Staubli VAL3: HOME.pjx

--- HOME.pjx ---
Parameters version=s7.7 stackSize=5000 millimeterUnit=true
Program file=checkPoint.pgx
Program file=checkZone.pgx
Program file=computeFrame.pgx
Program file=delete.pgx
Program file=deleteItem.pgx
Program file=duplicate.pgx
Program file=find.pgx
Program file=findMove.pgx
Program file=get.pgx
Program file=getDistance.pgx
Program file=getFrame.pgx
Program file=getFrameId.pgx
Program file=getFunctionEdit.pgx
Program file=getFunctionSel.pgx
Program file=getFunctionView.pgx
Program file=getJointData.pgx
Program file=getListItem.pgx
Program file=getMoveType.pgx
Program file=getPoint.pgx
Program file=getPointData.pgx
Program file=getSize.pgx
Program file=getSizeItem.pgx
Program file=getTool.pgx
Program file=getTrajItem.pgx
Program file=getTrajType.pgx
Program file=goTo.pgx
Program file=HerePoint.pgx
Program file=insertItem.pgx
Program file=insertValue.pgx
Program file=interpolateJ.pgx
Program file=link_me.pgx
Program file=listAdd.pgx
Program file=load.pgx
Program file=loadCycle.pgx
Program file=loadJoint.pgx
Program file=loadPage.pgx
Program file=loadPoint.pgx
Program file=makeTraj.pgx
Program file=moveTo.pgx
Program file=new.pgx
Program file=onEdit.pgx
Program file=onEditItem.pgx
Program file=onFunctionEdit.pgx
Program file=onFunctionSel.pgx
Program file=onFunctionView.pgx
Program file=onInsert.pgx
Program file=onProgEnd.pgx
Program file=onRun.pgx
Program file=onSave.pgx
Program file=onStart.pgx
Program file=onStop.pgx
Program file=orderDistance.pgx
Program file=orderZone.pgx
Program file=page_changeTrsf.pgx
Program file=scan_bestFit.pgx
Program file=select.pgx
Program file=selectProg.pgx
Program file=selectZone.pgx
Program file=setFrameId.pgx
Program file=setPointFrame.pgx
Program file=setTool.pgx
Program file=setTrajItem.pgx
Data file=HOME.dtx
Library alias=saveData path=Disk://saveData/saveData.pjx
Library alias=page path=Disk://kernel/template/page/page.pjx
Library alias=use path=Disk://kernel/userPage/userPage.pjx
Library alias=cycleStatus path=Disk://cycleStatus/cycleStatus.pjx
Library alias=language path=Disk://kernel/language/language.pjx
Library alias=tcp path=Disk://kernel/tool/tool.pjx
Library alias=prog path=Disk://instruction/PROG/PROG.pjx
Library alias=processList path=Disk://kernel/processList/processList.pjx
Library alias=solid path=Disk://trajectory/check_solid/check_solid.pjx
Library alias=pt path=Disk://kernel/template/session/saveTraj/HOME/HOME.pjx
Type name=TrajectoryItem path=Disk://kernel/template/TrajectoryItem/TrajectoryItem.pjx
Type name=ActionItem path=Disk://kernel/template/ActionItem/ActionItem.pjx
Type name=InstrItem path=Disk://kernel/template/InstrItem/InstrItem.pjx
Type name=Trajectory path=Disk://kernel/template/Trajectory/Trajectory.pjx
Type name=trajectoryType path=Disk://kernel/template/trajectory/trajectory.pjx
Type name=TrajHome path=Disk://kernel/template/TrajHome/TrajHome.pjx
Type name=TrajJoint path=Disk://kernel/template/TrajJoint/TrajJoint.pjx
Type name=TrajPoint path=Disk://kernel/template/TrajPoint/TrajPoint.pjx
Type name=FrameItem path=Disk://kernel/template/FrameItem/FrameItem.pjx

--- HOME.dtx ---
InstrItem tcpInstr
  [0]
    string sType
    string sData
Trajectory tTraj
  [0]
    TrajectoryItem tSuper[3]
      [0]
        num distance
        num moveType
        num nTime
        num nStop
        num nTcpAction
        string comment
        bool toStop
        mdesc nom_speed = {tmax=300, rmax=9999, leave=30, reach=30}
        InstrItem iInstr[3]
          [0]
            string sType
            string sData
          [1]
            string sType
            string sData
          [2]
            string sType
            string sData
        num nMoveId
      [1]
        num distance
        num moveType
        num nTime
        num nStop
        num nTcpAction
        string comment = "@JPOINT jZone1"
        bool toStop
        mdesc nom_speed = {tmax=9999, rmax=9999, leave=30, reach=30}
        InstrItem iInstr[3]
          [0]
            string sType
            string sData
          [1]
            string sType
            string sData
          [2]
            string sType
            string sData
        num nMoveId
      [2]
        num distance
        num moveType = 1
        num nTime
        num nStop
        num nTcpAction
        string comment = "@JPOINT jZone1Out"
        bool toStop
        mdesc nom_speed = {vel=450, tmax=1500, rmax=9999, leave=30, reach=30}
        InstrItem iInstr[3]
          [0]
            string sType
            string sData
          [1]
            string sType
            string sData
          [2]
            string sType
            string sData
        num nMoveId
    string sID = "HOME Zone1"
    num nId
public bool bMoveType[3]
  [0] = true
  [1] = true
public bool bStepping
bool bToSave
frame fFrame = {fatherId=world[0]}
frame fSetFrame = {x=-364.286321, y=-1043.316491, z=11.196424, rx=-6.99985, ry=11.31473, rz=18.24134, fatherId=world[0]}
mdesc nom_speed = {accel=25, vel=25, decel=25, blend=off}
num nCoeff = 1
num nDistance = 357.24033
num nHome
num nIndex
num nJoint
num nKey
num nSelected
num nView
num nZeta
pointRx pBestFit[3]
  [0] = {fatherId=world[0]}
  [1] = {fatherId=world[0]}
  [2] = {fatherId=world[0]}
pointRx pCheck = {fatherId=world[0]}
pointRx pNull = {fatherId=world[0]}
pointRx pPointTo = {fatherId=world[0]}
pointRx pPoints[3]
  [0] = {x=-364.286321, y=-1043.316491, z=11.196424, rx=84.453459, ry=18.310573, rz=168.800057, shoulder=lefty, elbow=epositive, wrist=wnegative, fatherId=world[0]}
  [1] = {x=-169.661081, y=-983.133224, z=-35.427424, rx=84.45454, ry=18.311675, rz=168.800636, shoulder=lefty, elbow=epositive, wrist=wnegative, fatherId=world[0]}
  [2] = {x=-263.249747, y=-701.832631, z=-51.099539, rx=84.453256, ry=18.310748, rz=168.801333, shoulder=lefty, elbow=epositive, wrist=wnegative, fatherId=world[0]}
string sInstruction
string sInstruction2
public string sItems[7]
  [0] = "cube_Salle_Bl"
  [1] = "cube_evac_rebut"
  [2] = "cube_moule"
  [3] = "cube_prelev"
  [4] = "home"
string sJoint = "Pt_Pass_Centre"
string sJointCycle = "Pt_Pass_Centre"
string sList
string sMessage
string sPoint = "Centre_Moule"
string sPointCycle = "Centre_Moule"
string sTrajType = "HOME"
trsf tAppro
trsf tPointTo
mdesc mMdesc = {accel=10, vel=10, decel=10, blend=off}
TrajHome jEditPoint
  [0]
    num nIndexTool
    TrajJointItem tData
      [0]
        jointRx jJoint
        TrajectoryItem tSuper
          [0]
            num distance
            num moveType
            num nTime
            num nStop
            num nTcpAction
            string comment
            bool toStop
            mdesc nom_speed = {accel=50, vel=50, decel=50, tmax=300, rmax=9999, leave=30, reach=30}
            InstrItem iInstr[3]
              [0]
                string sType
                string sData
              [1]
                string sType
                string sData
              [2]
                string sType
                string sData
            num nMoveId
    string sID
    num nZoneType
    num nZoneMove
    pointRx pO
    pointRx pX
    pointRx pY
    num nDimension
    pointRx pPointMove
    frame fFrame
    string sProgram
    num nIndexFrame
string sTrajCycle

--- checkPoint.pgx ---
public program checkPoint(point x_PointToGo (dimensions=1), point x_PointStart (dimensions=1), bool& x_bUnreached[] (dimensions=1), tool x_tTool (dimensions=1), bool x_bLinear (dimensions=1))
  local joint jPoint
  local string message
  local num i
  local trsf t
begin
  // check if the point is null
  if (cycleStatus:bCycle==false and cycleStatus:bSimulation==false) or !x_bLinear
    x_bUnreached=false
    t=position(x_PointToGo,world)
    if t!={0,0,0,0,0,0}
      //
      // look if the point that you want to reach is valid
      if x_bLinear
        //
        // use the percentage....
        //
        for i=0.1 to 1 step 0.1
          pCheck.trsf=interpolateL(position(x_PointStart,world),position(x_PointToGo,world),i)
          x_bUnreached=!pointToJoint(x_tTool,herej(),pCheck,jPoint)
          if x_bUnreached
            return
          endIf
        endFor
      else
        // joint move or check only the working area
        x_PointToGo.config={sfree,efree,wfree}
        x_bUnreached=!pointToJoint(x_tTool,herej(),x_PointToGo,jPoint)
      endIf
    endIf
  endIf
end

--- checkZone.pgx ---
program checkZone(point& x_pPoints[] (dimensions=1), tool x_tTool (dimensions=1), num x_nDimension (dimensions=1), num x_nType (dimensions=1), bool& x_bInside (dimensions=1))
begin
  // init the variable
  x_bInside=false
  // show the frame
  switch x_nType
    case 1
      //
      // BOX
      //
      //create the cube
      call solid:create_cube(x_pPoints[0],x_pPoints[1],x_pPoints[2],x_nDimension)
      // check the cube
      call solid:check_cube(x_tTool,x_bInside)
    break
    case 2
      //
      // SPHERE
      //
      // create the sphere
      call solid:create_sphere(x_pPoints,x_nDimension)
      // check the cube
      call solid:check_sphere(x_tTool,x_bInside)
    break
    case 3
      //
      // PLANE
      //
      //create the plane
      call solid:create_plane(x_pPoints[0],x_pPoints[1],x_pPoints[2])
      // check the cube
      call solid:check_plane(x_tTool,x_bInside)
    break
  endSwitch
end

--- delete.pgx ---
public program delete(string x_sName, num& x_nResult[])
  local string l_sItem
  local num l_nSize
  local string l_sMessage
begin
  //
  // delete the select trajectory
  //
  if isDefined(pt:tTraj[x_sName]) and x_sName!="home"
    // delete
    delete(pt:tTraj[x_sName])
    // save it
    bToSave=true
    x_nResult=0
  elseIf x_sName=="home"
    call language:message(l_sMessage,133)
    popUpMsg(l_sMessage)
  else
    x_nResult=-1
  endIf
end

--- findMove.pgx ---
program findMove(num x_nIndex, tool x_tTool, num& x_nMoveType[])
  local point l_pHere
  local num l_nResult
  local num l_nIndexTool
  local num l_nSize
  local num l_nMoveType
  local point l_pPoint[2]
  local joint l_jHere
  local bool l_bUnreach
begin
  //
  // MOVE TO THE POINT
  //
  // use the flange
  x_tTool=flange
  // get all the value that you need
  l_nSize=size(jEditPoint.tData)
  l_pHere=here(x_tTool,world)
  // get the point and the circle point
  call getPoint(l_pPoint,false,x_nIndex)
  pPoints[1].trsf=position(l_pPoint,world)
  pPoints[2].trsf={0,0,0,0,0,0}
  // Set to JOINT for default
  x_nMoveType=0
  // get the move TYPE
  call getMoveType(l_nMoveType,x_nIndex,false)
  //
  // move forward
  //
  if x_nIndex>0 and l_nMoveType==1
    // get the point and the circle point
    call getPoint(l_pPoint,false,x_nIndex-1)
    pPoints.trsf=position(l_pPoint,world)
    if distance(l_pHere,pPoints)<25
      // set to linear
      x_nMoveType=1
    elseIf setFrame(pPoints,pPoints[1],pPoints[2],fSetFrame)==0
      // check frame
      l_pHere=here(x_tTool,fSetFrame)
      pPoints[1].trsf=position(pPoints[1],fSetFrame)
      if l_pHere.trsf.x>=0 and l_pHere.trsf.x<=pPoints[1].trsf.x and abs(l_pHere.trsf.y)<10 and abs(l_pHere.trsf.z)<10
        // set to linear
        x_nMoveType=1
      endIf
    endIf
  endIf
  //
  // move back
  //
  if x_nIndex<(l_nSize-1) and x_nMoveType!=1
    call getMoveType(l_nMoveType,x_nIndex+1,false)
    if l_nMoveType==1
      // get the point and the circle point
      call getPoint(l_pPoint,false,x_nIndex)
      pPoints[1].trsf=position(l_pPoint,world)
      // get the point and the circle point
      call getPoint(l_pPoint,false,x_nIndex+1)
      pPoints.trsf=position(l_pPoint,world)
      if distance(l_pHere,pPoints)<25
        // switch to linear
        x_nMoveType=1
      elseIf setFrame(pPoints,pPoints[1],pPoints[2],fSetFrame)==0
        // check frame
        l_pHere=here(x_tTool,fSetFrame)
        pPoints[1].trsf=position(pPoints[1],fSetFrame)
        if l_pHere.trsf.x>=0 and l_pHere.trsf.x<=pPoints[1].trsf.x and abs(l_pHere.trsf.y)<10 and abs(l_pHere.trsf.z)<10
          // set to linear
          x_nMoveType=1
        endIf
      endIf
    endIf
  endIf
end

--- getFrame.pgx ---
public program getFrame(frame& x_fFrame[], bool x_bCycle)
  local num l_nIndex
begin
  // CYCLE
  if x_bCycle
    l_nIndex=pt:tTraj[sTrajCycle].nIndexFrame
  else
    // NOT CYCLE
    l_nIndex=jEditPoint.nIndexFrame
  endIf
  x_fFrame.trsf=saveData:fFrameItem[l_nIndex].fFrame.trsf
end

--- getFrameId.pgx ---
public program getFrameId(num& x_nFrame)
begin
  // give back the frame
  x_nFrame=jEditPoint.nIndexFrame
end

--- getFunctionEdit.pgx ---
public program getFunctionEdit(string& x_sName[])
  local string l_sMessage
begin
  //
  // define your message for the
  // function KEY
  //
  // NOTE is an ARRAY[0..7]
  //
  // example:
  // x_sName[1]="DEMO"
  // active the F2 button
  //
  if (nIndex>0 or jEditPoint.nZoneType==0) and find(jEditPoint.tData[nIndex].tSuper.comment,"@")==-1
    // here
    call language:message(l_sMessage,150)
    x_sName[0]=l_sMessage
  else
  // ALIGN
  call language:message(l_sMessage,134)
  x_sName[1]=l_sMessage
  // Tool
  call language:message(l_sMessage,123)
  x_sName[2]=l_sMessage
  endIf
//  // define the @Link
//  x_sName[1]="@Link"
end

--- getFunctionSel.pgx ---
public program getFunctionSel(string& x_sName[])
  local string l_sMessage
begin
  //
  // define your message for the
  // function KEY
  //
  // NOTE is an ARRAY[0..7]
  //
  // example:
  // x_sName[1]="DEMO"
  // active the F2 button
  //
  // Set Home Program
  call language:message(l_sMessage,135)
  x_sName[2]=l_sMessage
  call language:message(l_sMessage,136)
  x_sName[3]=l_sMessage
end

--- getFunctionView.pgx ---
public program getFunctionView(string& x_sName[])
  local string l_sMessage
begin
  //
  // define your message for the
  // function KEY
  //
  // NOTE is an ARRAY[0..7]
  //
  // example:
  // x_sName[1]="DEMO"
  // active the F2 button
  //
  // define the @Link
  // here
  call language:message(l_sMessage,150)
  x_sName[0]=l_sMessage
  // x_sName[1]="@Link"
    // ALIGN
  call language:message(l_sMessage,134)
  x_sName[1]=l_sMessage
end

--- getJointData.pgx ---
public program getJointData(joint& x_jJoint, tool& x_tTool, bool x_bCycle, num x_nIndex)
  local point l_pPoint
  local num l_nSize
  local string l_sName
  local num l_nResult
  local string l_sComment
  local num l_nType
  local point l_pPointTo
  local num i
begin
  //
  //   !!! REMOVE DUE PROBLEMS of CROSS LINK
  //
  //   get the comment type
  //    if x_bCycle
  //      l_sComment=pt:tTraj[sTrajCycle].tData[x_nIndex].tSuper.comment
  //    else
  //      l_sComment=jEditPoint.tData[x_nIndex].tSuper.comment
  //    endIf
  //    if find(l_sComment,"@POINT")!=-1
  //      //
  //      // POINT
  //      //
  //      l_sName=right(l_sComment,len(l_sComment)-len("@POINT "))
  //      call loadPoint(l_sName,l_nResult)
  //      if l_nResult==0
  //        // use the flange
  //        x_tTool=flange
  //        // get the tool
  //        //call tcp:getTool(x_tTool,pPoint:tTraj[l_sName].nIndexTool)
  //        // get the last point using the depart point
  //        l_nSize=size(pPoint:tTraj[l_sName].tData)
  //        // find the point use the real one
  //        for i=0 to l_nSize-1
  //          l_nType=pPoint:tTraj[l_sName].tData[i].nType
  //          if l_nType==1
  //            // get the real point
  //            l_pPointTo=pPoint:tTraj[l_sName].tData[i].pPoint
  //          endIf
  //        endFor
  //        // take the DEPART
  //        l_pPoint=pPoint:tTraj[l_sName].tData[l_nSize-1].pPoint
  //        l_pPoint=appro(l_pPointTo,l_pPoint.trsf)
  //        // give back
  //        pointToJoint(x_tTool,herej(),l_pPoint,x_jJoint)
  //      endIf
  //    elseIf find(l_sComment,"@JPOINT")!=-1
  //      //
  //      // JPOINT
  //      //
  //      l_sName=right(l_sComment,len(l_sComment)-len("@JPOINT "))
  //      call loadJoint(l_sName,l_nResult)
  //      if l_nResult==0
  //        // use the flange
  //        x_tTool=flange
  //        // give back
  //        //call tcp:getTool(x_tTool,jPoint:tTraj[l_sName].nIndexTool)
  //        x_jJoint=jPoint:tTraj[l_sName].tData[0].jJoint
  //      endIf
  //    else
  // give back
  // use the flange
  x_tTool=flange
  if x_bCycle
    x_jJoint=pt:tTraj[sTrajCycle].tData[x_nIndex].jJoint
    //      call tcp:getTool(x_tTool,pt:tTraj[sTrajCycle].nIndexTool)
  else
    x_jJoint=jEditPoint.tData[x_nIndex].jJoint
    //      call tcp:getTool(x_tTool,jEditPoint.nIndexTool)
  endIf
  //endIf
  if l_nResult!=0
    // remove the link
    jEditPoint.tData[x_nIndex].tSuper.comment=""
  endIf
end

--- getListItem.pgx ---
public program getListItem(string& x_sItem[], num x_nIndex)
  local string l_sItem4[4]
  local string l_sZoneType
  local string l_sZoneMove
  local string l_sItem7[7]
  local joint l_jJoint
  local tool l_tTool
  local string l_sItem[6]
begin
  //
  // define the item to show in the edit page Traj
  // customize an array and copy to x_sItem...
  //
  // see other traj as example
  l_sItem[0]=l_sItem7[0]=("Joint 1 > "+toString(".2",jEditPoint.tData[x_nIndex].jJoint.j1))
  l_sItem[1]=l_sItem7[1]=("Joint 2 > "+toString(".2",jEditPoint.tData[x_nIndex].jJoint.j2))
  l_sItem[2]=l_sItem7[2]=("Joint 3 > "+toString(".2",jEditPoint.tData[x_nIndex].jJoint.j3))
  l_sItem[3]=l_sItem7[3]=("Joint 4 > "+toString(".2",jEditPoint.tData[x_nIndex].jJoint.j4))
  l_sItem[4]=l_sItem7[4]=("Joint 5 > "+toString(".2",jEditPoint.tData[x_nIndex].jJoint.j5))
  l_sItem[5]=l_sItem7[5]=("Joint 6 > "+toString(".2",jEditPoint.tData[x_nIndex].jJoint.j6))
  call use:stringCopy(l_sItem,x_sItem)
  switch x_nIndex
    case 0
      // add_on for the zone definition
      switch jEditPoint.nZoneType
        case 1
          l_sZoneType=" > Box"
        break
        case 2
          l_sZoneType=" > Sphere"
        break
        case 3
          l_sZoneType=" > Plane"
        break
        default
          l_sZoneType=" > "
        break
      endSwitch
      // show only the necessary
      if jEditPoint.nZoneType[x_nIndex]==0
        l_sItem7[6]=("Zone "+l_sZoneType)
        call use:stringCopy(l_sItem7,x_sItem)
      else
        // only the move type
        l_sItem4[0]=("Zone "+l_sZoneType)
        switch jEditPoint.nZoneMove
          case 0
            l_sZoneMove="Point"
          break
          case 1
            l_sZoneMove="Appro"
          break
          case 2
            l_sZoneMove="Z Value"
          break
          case 3
            l_sZoneMove="@Point"
          break
          case 4
            l_sZoneMove="@JPoint"
          break
        endSwitch
        l_sItem4[1]="  └───>[EDIT] "
        l_sItem4[2]=("MoveTO > "+l_sZoneMove)
        if (jEditPoint.nZoneMove==3 or jEditPoint.nZoneMove==4) and find(jEditPoint.tData.tSuper.comment,"@")!=-1
          l_sItem4[3]="  └> "+jEditPoint.tData.tSuper.comment
        else
          l_sItem4[3]="  └───>[EDIT] "
        endIf
        // insert all
        call use:stringCopy(l_sItem4,x_sItem)
      endIf
    break
    default
      // insert only the coordinate
      call use:stringCopy(l_sItem,x_sItem)
    break
  endSwitch
  // save the actual index
  nIndex=x_nIndex
end

--- getMoveType.pgx ---
public program getMoveType(num& x_nMoveType[], num x_nIndex, bool x_bCycle)
begin
  // get the moveType
  if x_bCycle
    x_nMoveType=pt:tTraj[sTrajCycle].tData[x_nIndex].tSuper.moveType
  else
    x_nMoveType=jEditPoint.tData[x_nIndex].tSuper.moveType
  endIf
end

--- getPoint.pgx ---
public program getPoint(point& x_pPoint[] (dimensions=1), bool x_bCycle (dimensions=1), num x_nIndex (dimensions=1))
  local string l_sItem
  local tool l_tTool
  local joint l_jJoint
begin
  // check the point
  link(x_pPoint,world)
  // use the flange
  l_tTool=flange
  // give back the point
  call getJointData(l_jJoint,l_tTool,x_bCycle,x_nIndex)
  x_pPoint=jointToPoint(l_tTool,world,l_jJoint)
end

--- getPointData.pgx ---
program getPointData(num& x_nSpeed[], mdesc& x_mDesc[], num& x_nDistance[], bool& x_bToStop[], num& x_nMoveType[], num& x_nStop[], num x_nIndex, bool x_bCycle)
begin
  if x_bCycle
    // get tha parameter
    // SPEED
    // get the speed in mm/sec
    if pt:tTraj[sTrajCycle].tData[x_nIndex].tSuper.moveType==0
      x_nSpeed=pt:tTraj[sTrajCycle].tData[x_nIndex].tSuper.nom_speed.vel*15
    else
      if pt:tTraj[sTrajCycle].tData[x_nIndex].tSuper.moveType==1
        x_nSpeed=pt:tTraj[sTrajCycle].tData[x_nIndex].tSuper.nom_speed.tvel
      endIf
    endIf
    // MDESC
    x_mDesc=pt:tTraj[sTrajCycle].tData[x_nIndex].tSuper.nom_speed
    // DISTANCE
    x_nDistance=pt:tTraj[sTrajCycle].tData[x_nIndex].tSuper.distance
    //  check  for a stop using
    x_bToStop=pt:tTraj[sTrajCycle].tData[x_nIndex].tSuper.toStop
    // get MoveType
    x_nMoveType=pt:tTraj[sTrajCycle].tData[x_nIndex].tSuper.moveType
  else
    // get tha parameter
    // SPEED
    // get the speed in mm/sec
    if jEditPoint.tData[x_nIndex].tSuper.moveType==0
      x_nSpeed=jEditPoint.tData[x_nIndex].tSuper.nom_speed.vel*15
    else
      if jEditPoint.tData[x_nIndex].tSuper.moveType==1
        x_nSpeed=jEditPoint.tData[x_nIndex].tSuper.nom_speed.tvel
      endIf
    endIf
    // MDESC
    x_mDesc=jEditPoint.tData[x_nIndex].tSuper.nom_speed
    // DISTANCE
    x_nDistance=jEditPoint.tData[x_nIndex].tSuper.distance
    //  check  for a stop using
    x_bToStop=jEditPoint.tData[x_nIndex].tSuper.toStop
    // get MoveType
    x_nMoveType=jEditPoint.tData[x_nIndex].tSuper.moveType
  endIf
end

--- getSize.pgx ---
public program getSize(num& x_nSize[])
  local string l_sType
begin
  // give back the size to trajectory field
  x_nSize=size(pt:tTraj)
end

--- getTool.pgx ---
public program getTool(num& x_nTool)
begin
  //
  // get the tool
  //
  x_nTool=jEditPoint.nIndexTool
end

--- getTrajItem.pgx ---
public program getTrajItem(TrajectoryItem& x_tTrajItem[], num x_nIndex)
begin
  //
  // get all the FIELD
  //
  x_tTrajItem=jEditPoint.tData[x_nIndex].tSuper
end

--- getTrajType.pgx ---
program getTrajType(string& x_sTrajType[])
  local num l_nPos
  local string l_sPath
begin
  // get the trajType
  l_sPath=libPath()
  if find(l_sPath,sTrajType)==-1
    do
      l_nPos=find(l_sPath,"/")
      if l_nPos==-1
        l_nPos=find(l_sPath,"\")
      endIf
      if l_nPos!=-1
        l_sPath=right(l_sPath,len(l_sPath)-l_nPos-1)
      endIf
    until l_nPos==-1
    //
    sTrajType=l_sPath
  endIf
  // return back
  x_sTrajType=sTrajType
end

--- goTo.pgx ---
public program goTo(tool x_tTool, mdesc x_mDesc, num x_nMoveType, bool& x_bUnreached[], num x_nIndex)
  local mdesc temp_mdesc
  local num l_nSize
  local point l_pPoint
  local joint l_jJoint
  local frame l_ZoneFrame
  local bool l_bCheck
  local num l_nType
  local num l_nDimension
  local tool l_tTool
  local string l_sMessage
  local num l_nMoveId
begin
  // check for the zone
  if (jEditPoint.nZoneType!=0 and x_nIndex==0) or find(jEditPoint.tData[x_nIndex].tSuper.comment,"@")!=-1
    // take the tool
    // use flange
    l_tTool=flange
    //call tcp:getTool(l_tTool,jEditPoint.nIndexTool)
    // take the three points
    pPoints[0]=jEditPoint.pO
    pPoints[1]=jEditPoint.pX
    pPoints[2]=jEditPoint.pY
    // take the distance
    l_nDimension=jEditPoint.nDimension
    //take the type
    l_nType=jEditPoint.nZoneType
    // check the frame type-2 CIRCLE
    if setFrame(pPoints[0],pPoints[1],pPoints[2],fSetFrame)==0 or l_nType==2
      call checkZone(pPoints,l_tTool,l_nDimension,l_nType,l_bCheck)
      // show the result
      if l_bCheck
        // inside the zone
        call language:message(l_sMessage,225)
        // move TO
        call moveTo(l_tTool,x_mDesc,x_nMoveType,x_bUnreached,x_nIndex,l_nMoveId,false)
      elseIf find(jEditPoint.tData[x_nIndex].tSuper.comment,"@")!=-1
        // link POINT
        // look for the moveType
        call findMove(x_nIndex,l_tTool,x_nMoveType)
        call moveTo(l_tTool,x_mDesc,x_nMoveType,x_bUnreached,x_nIndex,l_nMoveId,false)
      else
        //outside the zone
        call language:message(l_sMessage,226)
      endIf
    elseIf find(jEditPoint.tData[x_nIndex].tSuper.comment,"@")!=-1
      // found a @POINT-JPOINT
      call moveTo(l_tTool,x_mDesc,x_nMoveType,x_bUnreached,x_nIndex,l_nMoveId,false)
    else
      // frame not define
      call language:message(l_sMessage,183)
      call use:timerDialog(l_sMessage,3)
    endIf
  elseIf isInRange(jEditPoint.tData[x_nIndex].jJoint)
    // look for the moveType
    call findMove(x_nIndex,x_tTool,x_nMoveType)
    // execute the movement
    switch x_nMoveType
      case 0
        // JOINT MOVE
        // go to the select Joint
        movej(jEditPoint.tData[x_nIndex].jJoint,x_tTool,x_mDesc)
      break
      case 1
        // LINEAR MOVE
        movel(jointToPoint(x_tTool,world,jEditPoint.tData[x_nIndex].jJoint),x_tTool,x_mDesc)
      break
      default
      break
    endSwitch
  else
    x_bUnreached=true
  endIf
  // save the actual index
  nIndex=x_nIndex
end

--- insertValue.pgx ---
program insertValue(num& x_nValue[] (dimensions=1), num x_nIndex (dimensions=1))
begin
  if nDistance[0]!=-1
    // insert
    insert(nDistance[x_nIndex])
    insert(nCoeff[x_nIndex])
    insert(nJoint[x_nIndex])
    insert(nHome[x_nIndex])
  endIf
  // copy
  nCoeff[x_nIndex]=x_nValue[3]
  nDistance[x_nIndex]=x_nValue[2]
  nJoint[x_nIndex]=x_nValue[1]
  nHome[x_nIndex]=x_nValue
end

--- interpolateJ.pgx ---
public program interpolateJ(joint p_j1, joint p_j2, num p_nInterpolate, joint& x_jRetVal[], bool& x_bRetVal[])
begin
  // Interpolierten Jointwert berechnen
  x_jRetVal.j1=(p_j2.j1-p_j1.j1)*p_nInterpolate+p_j1.j1
  x_jRetVal.j2=(p_j2.j2-p_j1.j2)*p_nInterpolate+p_j1.j2
  x_jRetVal.j3=(p_j2.j3-p_j1.j3)*p_nInterpolate+p_j1.j3
  x_jRetVal.j4=(p_j2.j4-p_j1.j4)*p_nInterpolate+p_j1.j4
  x_jRetVal.j5=(p_j2.j5-p_j1.j5)*p_nInterpolate+p_j1.j5
  x_jRetVal.j6=(p_j2.j6-p_j1.j6)*p_nInterpolate+p_j1.j6
  x_bRetVal=isInRange(x_jRetVal)
end

--- link_me.pgx ---
program link_me(num x_nIndex)
  local num i
  local num l_nSize
  local string l_sItem
  local num l_nKey
  local num l_nIndex
  local string l_sEvent
begin
  //
  // !!! REMOVE DUE PROBLEMS of CROSS LINK
  //
  //  // @POINT -> use depart
  //  // @JOINT -> use the first JOINT
  //  call use:clear(0,13)
  //  call use:type(5,13,"@Link")
  //  call use:setSizeList(4,8,8,3)
  //  call use:listcreate("")
  //  l_sItem=" NONE "
  //  call use:listadd(l_sItem)
  //  l_sItem="@JPOINT"
  //  call use:listadd(l_sItem)
  //  //  l_sItem="@POINT"
  //  //  call use:listadd(l_sItem)
  //  // refresh it
  //  call use:listupdate(0)
  //  // get the item
  //  do
  //    l_nKey=get()
  //    call use:listevent(l_nKey,l_nIndex,l_sEvent)
  //  until l_nKey==270 or l_nKey==255
  //  if l_nKey==270
  //    // select the @Point - @jPoint
  //    // build the list
  //    call use:setSizeList(0,0,16,12)
  //    switch l_nIndex
  //      case 2
  //        call use:listcreate("@Point")
  //        // insert all the item
  //        l_sItem=first(pPoint:tTraj)
  //        call use:listadd(l_sItem)
  //        // search it
  //        while l_sItem!=""
  //          l_sItem=next(pPoint:tTraj[l_sItem])
  //          call use:listadd(l_sItem)
  //        endWhile
  //        l_sItem="@POINT "
  //      break
  //      case 1
  //        call use:listcreate("@JPoint")
  //        // insert all the item
  //        l_sItem=first(jPoint:tTraj)
  //        call use:listadd(l_sItem)
  //        // search it
  //        while l_sItem!=""
  //          l_sItem=next(jPoint:tTraj[l_sItem])
  //          call use:listadd(l_sItem)
  //        endWhile
  //        l_sItem="@JPOINT "
  //      break
  //      case 0
  //        // empty one
  //        l_sItem=l_sEvent=""
  //      break
  //    endSwitch
  //    if l_nIndex!=0
  //      // refresh it
  //      call use:listupdate(0)
  //      // get the item
  //      do
  //        l_nKey=get()
  //        call use:listevent(l_nKey,l_nIndex,l_sEvent)
  //      until l_nKey==270 or l_nKey==255
  //    endIf
  //    // give back
  //    if l_nKey==270
  //      // save it
  //      jEditPoint.tData[x_nIndex].tSuper.comment=l_sItem+l_sEvent
  //      if x_nIndex==0
  //        jEditPoint.nZoneType=0
  //      endIf
  //    endIf
  //  endIf
end

--- load.pgx ---
public program load(string x_sItem, num& x_nResult)
  local string l_sType
  local string l_sPath
  local string l_sMessage
begin
  // load the select trajectory..already loaded
  call getTrajType(l_sType)
  if find(pt:libPath(),saveData:sPathTraj)==-1
    pt:libLoad(saveData:sPathTraj+l_sType)
    delay(0)
    if saveData:bDebug
      ? "loading HOME..."+saveData:sPathTraj+l_sType
    endIf
  endIf
  if isDefined(pt:tTraj[x_sItem])
    // use the type...
    call pt:link_it(x_sItem)
    jEditPoint=pt:tTraj[x_sItem]
    jEditPoint.sID=x_sItem
    x_nResult=0
  elseIf x_sItem!=""
    // not FOUND
    call language:message(l_sMessage,-7)
    x_nResult=-1
    popUpMsg(l_sMessage+x_sItem)
    jEditPoint.sID=""
  elseIf x_sItem==""
    // reload all the template
    call loadJoint("",x_nResult)
    call loadPoint("",x_nResult)
  endIf
end

--- loadCycle.pgx ---
public program loadCycle(string x_sItem, num& x_nResult[])
  local string l_sType
  local string l_sPath
begin
  // load the select trajectory..already loaded
  call getTrajType(l_sType)
  if find(pt:libPath(),saveData:sPathTraj)==-1
    pt:libLoad(saveData:sPathTraj+l_sType)
    delay(0)
  endIf
  if isDefined(pt:tTraj[x_sItem])
    // use the type...
    call pt:link_it(x_sItem)
    sTrajCycle=x_sItem
  else
    x_nResult=-1
  endIf
end

--- loadJoint.pgx ---
public program loadJoint(string x_sItem, num& x_nResult)
  local string l_sType
  local string l_sMessage
  local num l_nResult
begin
  //
  // !!! REMOVE DUE PROBLEMS of CROSS LINK
  //
  //
  //  // load the select trajectory..already loaded
  //  call getTrajType(l_sType)
  //  if find(jPoint:libPath(),saveData:sPathTraj)==-1
  //    l_nResult=jPoint:libLoad(saveData:sPathTraj+"JPOINT")
  //    delay(0)
  //    if saveData:bDebug
  //      ? "HOME loading JPOINT..."+saveData:sPathTraj+"JPOINT"+toString("",l_nResult)
  //    endIf
  //  endIf
  //  if isDefined(jPoint:tTraj[x_sItem])
  //    // validate
  //    x_nResult=0
  //  elseIf x_sItem!=""
  //    // not FOUND
  //    call language:message(l_sMessage,-7)
  //    x_nResult=-1
  //    popUpMsg(l_sMessage+x_sItem)
  //  endIf
end

--- loadPage.pgx ---
program loadPage(string x_sPage, string& x_sItems[])
// load the next page
  local num i
begin
  // look if the page libload is correct
  i=page:libLoad(x_sPage)
  delay(0)
  logMsg("KERNEL:PAGE LIBLOAD "+x_sPage+" result "+toString("",i))
  if i!=0
    popUpMsg("Loading page "+x_sPage+" error CODE "+toString("",i))
  else
    page:sItems=x_sItems
    call page:main()
  endIf
end

--- loadPoint.pgx ---
public program loadPoint(string x_sItem, num& x_nResult)
  local string l_sType
  local string l_sMessage
  local num l_nResult
begin
  //
  // !!! REMOVE DUE PROBLEMS of CROSS LINK
  //
  //  // load the select trajectory..already loaded
  //  call getTrajType(l_sType)
  //  if find(pPoint:libPath(),saveData:sPathTraj)==-1
  //    l_nResult=pPoint:libLoad(saveData:sPathTraj+"POINT")
  //    delay(0)
  //    if saveData:bDebug
  //      ? "HOME loading POINT..."+saveData:sPathTraj+"POINT"+toString("",l_nResult)
  //    endIf
  //  endIf
  //  if isDefined(pPoint:tTraj[x_sItem])
  //    // validate
  //    x_nResult=0
  //  elseIf x_sItem!=""
  //    // not FOUND
  //    call language:message(l_sMessage,-7)
  //    x_nResult=-1
  //    popUpMsg(l_sMessage+x_sItem)
  //  endIf
end

--- makeTraj.pgx ---
program makeTraj(num x_nJointStart, string x_sTrajLoad)
  local num i
  local bool l_bToStop[2]
  local num l_nSize
  local tool l_tTool
  local num l_nSpeed[2]
  local mdesc l_mDesc[2]
  local num l_nDistance[2]
  local num l_nMoveType[2]
  local point l_pAction
  local bool l_bUnreached
  local num l_nStop
  local point l_pCheck[3]
  local point l_pHere
  local frame l_fPlane
  local num l_nTime
  local string l_sType
  local string l_sMessage
  local bool l_bConnection
  local num l_nMoveId
  local TrajectoryItem l_tTraj
  local joint l_jJoint
  local ActionItem l_aAction
  local num j
  local bool l_bGoToCloseP
  local point l_pHereJ
  local joint l_jResult
  local bool l_bOk
  local num i_from
  local num i_to
  local joint l_jHere
  local joint l_jRunJoint[2]
begin
  //
  // inizialize the system
  //
  // use the flange
  l_tTool=flange
  // the maximum size
  call getSizeItem(true,l_nSize)
  //
  // first go near by straight line of the two previous points
  //
  if pt:tTraj[sTrajCycle].nZoneType!=0 and x_nJointStart==0
    // use of the ZONE TYPE
    switch pt:tTraj[sTrajCycle].nZoneMove
      case 0
        l_sType="POINT"
      break
      case 1
        l_sType="APPRO"
      break
      case 2
        l_sType="Z VALUE"
      break
      case 3
        l_sType="@Point"
      break
      case 4
        l_sType="@JPoint"
      break
    endSwitch
    cycleStatus:sToShow="Move using: "+l_sType+toString("",x_nJointStart)+"# of the home: "+x_sTrajLoad
    logMsg("HOMING: "+l_sMessage)
    call getPointData(l_nSpeed,l_mDesc,l_nDistance,l_bToStop,l_nMoveType,l_nStop,0,true)
    call moveTo(l_tTool,l_mDesc,l_nMoveType,l_bUnreached,0,l_nMoveId,true)
    waitEndMove()
    // set the start point
    x_nJointStart=1
  elseIf saveData:bUseHomeScanner
    // look FORWARD
    if x_nJointStart<l_nSize-1
      // get all the JOINT
      call getJointData(l_jRunJoint[0],l_tTool,true,x_nJointStart+1)
      call getJointData(l_jRunJoint[1],l_tTool,true,x_nJointStart)
      // look if there is
      if setFrame(jointToPoint(l_tTool,world,l_jRunJoint[0]),jointToPoint(l_tTool,world,l_jRunJoint[1]),pNull,fFrame)==0
        pCheck=here(l_tTool,fFrame)
        if pCheck.trsf.x>=0
          //
          // go to nearest point
          //
          call getPoint(l_pCheck[0],true,x_nJointStart+1)
          call getPoint(l_pCheck[1],true,x_nJointStart)
          x_nJointStart=x_nJointStart+1
          l_bGoToCloseP=true
        endIf
      endIf
    endIf
    // LOOK BACKWARD
    if !l_bGoToCloseP and x_nJointStart>0
      // get all the JOINT
      call getJointData(l_jRunJoint[0],l_tTool,true,x_nJointStart)
      call getJointData(l_jRunJoint[1],l_tTool,true,x_nJointStart-1)
      // look if there is
      if setFrame(jointToPoint(l_tTool,world,l_jRunJoint[0]),jointToPoint(l_tTool,world,l_jRunJoint[1]),pNull,fFrame)==0
        pCheck=here(l_tTool,fFrame)
        if pCheck.trsf.x>=0
          //
          // go to nearest point
          //
          call getPoint(l_pCheck[0],true,x_nJointStart)
          call getPoint(l_pCheck[1],true,x_nJointStart-1)
          l_bGoToCloseP=true
        endIf
      endIf
    endIf
    // go to an approach POINT
    if l_bGoToCloseP
      // init
      l_pCheck[2]=here(l_tTool,world)
      l_pHere=here(l_tTool,world)
      l_pHereJ=here(flange,world)
      l_nDistance=10000
      // check the nearest point
      l_nMoveType=pt:tTraj[sTrajCycle].tData[x_nJointStart].tSuper.moveType
      for i=0 to 1 step 0.1
        if l_nMoveType==0
          call interpolateJ(l_jRunJoint[1],l_jRunJoint[0],i,l_jResult,l_bOk)
          l_pCheck[2]=jointToPoint(flange,world,l_jResult)
          if l_nDistance>=distance(l_pCheck[2],l_pHereJ)
            l_nDistance=distance(l_pCheck[2],l_pHereJ)
            //save the value
            l_nStop=i
          endIf
        else
          l_pCheck[2].trsf=interpolateL(l_pCheck[1].trsf,l_pCheck[0].trsf,i)
          l_bOk=true
          if l_nDistance>=distance(l_pCheck[2],l_pHere)
            l_nDistance=distance(l_pCheck[2],l_pHere)
            //save the value
            l_nStop=i
          endIf
        endIf
      endFor
      // closer search
      i_from=(max(l_nStop-0.05,0))
      i_to=(min(l_nStop+0.05,1))
      for i=i_from to i_to step 0.01
        if l_nMoveType==0
          call interpolateJ(l_jRunJoint[1],l_jRunJoint[0],i,l_jResult,l_bOk)
          l_pCheck[2]=jointToPoint(flange,world,l_jResult)
          if l_nDistance>=distance(l_pCheck[2],l_pHereJ)
            l_nDistance=distance(l_pCheck[2],l_pHereJ)
            //save the value
            l_nStop=i
          endIf
        else
          l_pCheck[2].trsf=interpolateL(l_pCheck[1].trsf,l_pCheck[0].trsf,i)
          l_bOk=true
          if l_nDistance>=distance(l_pCheck[2],l_pHere)
            l_nDistance=distance(l_pCheck[2],l_pHere)
            //save the value
            l_nStop=i
          endIf
        endIf
      endFor
      // set the best one
      call getPointData(l_nSpeed,l_mDesc,l_nDistance,l_bToStop,l_nMoveType,l_nStop,x_nJointStart,true)
      l_jHere=herej()
      if l_nMoveType==0
        call interpolateJ(l_jRunJoint[1],l_jRunJoint[0],l_nStop,l_jResult,l_bOk)
        l_pCheck[2]=jointToPoint(flange,world,l_jResult)
        // put the wrist on free
        l_pCheck[2].config.wrist=wfree
        if pointToJoint(l_tTool,herej(),l_pCheck[2],l_jHere)
          movej(l_pCheck[2],flange,l_mDesc)
        endIf
      else
        l_pCheck[2].trsf=interpolateL(l_pCheck[1].trsf,l_pCheck[0].trsf,l_nStop)
        // put the wrist on free
        l_pCheck[2].config.wrist=wfree
        if pointToJoint(l_tTool,herej(),l_pCheck[2],l_jHere)
          movej(l_pCheck[2],l_tTool,l_mDesc)
        endIf
      endIf
      // show the message
      cycleStatus:sToShow="Move to point: "+toString("",x_nJointStart+1)+" of: "+x_sTrajLoad +" % "+toString(".3",l_nStop)
      logMsg("HOMING: "+cycleStatus:sToShow)
      waitEndMove()
    endIf
  endIf
  //
  // for all of my traj cyclePoints move the robot
  //
  resize(tTraj.tSuper,1,size(pt:tTraj[sTrajCycle].tData))
  for i=x_nJointStart to (l_nSize-1)
    tTraj.tSuper[i]=pt:tTraj[sTrajCycle].tData[i].tSuper
  endFor
  tTraj.sID="HOME "+pt:tTraj[sTrajCycle].sID
  call cycleStatus:addTraj(tTraj)
  // show the message
  cycleStatus:sToShow="Moving from point: "+toString("",x_nJointStart+1)+" of : "+x_sTrajLoad
  logMsg("HOMING: "+cycleStatus:sToShow)
  for i=x_nJointStart to (l_nSize-1)
    //
    // get the point info
    //
    l_tTraj=pt:tTraj[sTrajCycle].tData[i].tSuper
    //
    // get the distance in percentage
    //
    call getDistance(l_tTool,l_nDistance,true,i)
    //
    // give to the traj library the percentage distance
    //
    if l_tTraj.toStop
      l_tTraj.nom_speed.blend=off
    endIf
    //
    // put the move in the stack
    //
    l_jJoint=pt:tTraj[sTrajCycle].tData[i].jJoint
    call moveTo(l_tTool,l_tTraj.nom_speed,l_tTraj.moveType,l_bUnreached,i,l_nMoveId,true)
    // set the data
    l_aAction.nDistance=l_nDistance
    l_aAction.nPointId=i
    l_aAction.nMoveId=l_nMoveId
    l_aAction.sIdTraj="HOME "+pt:tTraj[sTrajCycle].sID
    call cycleStatus:putInstr_Traj(l_aAction,l_tTraj,pt:tTraj[sTrajCycle].nIndexTool,l_nSize)
    // there is a waitEndMove
    if l_tTraj.toStop
      waitEndMove()
      delay(l_tTraj.nStop)
      // wait all the action has been done
      wait(cycleStatus:bActionRunning==false)
    endIf
  endFor
end

--- moveTo.pgx ---
public program moveTo(tool x_tTool, mdesc x_mDesc, num x_nMoveType, bool& x_bUnreached[], num x_nIndex, num& x_nMoveId, bool x_bCycle)
  local frame l_fFrame
  local point l_pHere
  local point l_pMove
  local string l_sName
  local num i
  local num l_nType
  local num l_nIndex
  local num l_nResult
  local joint l_jMove
  local num l_nSize
  local tool l_tTool
  local point l_pPoint
begin
  if x_bCycle
    //
    // go to the select Joint
    //
    // use the go to the defined type...
    if x_nIndex==0 and pt:tTraj[sTrajCycle].nZoneType!=0
      switch pt:tTraj[sTrajCycle].nZoneMove
        // POINT TO
        case 0
          if x_nMoveType==0
            x_nMoveId=movej(pt:tTraj[sTrajCycle].pPointMove,x_tTool,x_mDesc)
          elseIf x_nMoveType==1
            x_nMoveId=movel(pt:tTraj[sTrajCycle].pPointMove,x_tTool,x_mDesc)
          endIf
        break
        case 1
          // APPRO use the real APPRO
          call tcp:getTool(l_tTool,pt:tTraj[sTrajCycle].nIndexTool)
          if x_nMoveType==0
            x_nMoveId=movej(appro(here(l_tTool,world),pt:tTraj[sTrajCycle].pPointMove.trsf),x_tTool,x_mDesc)
          elseIf x_nMoveType==1
            x_nMoveId=movel(appro(here(l_tTool,world),pt:tTraj[sTrajCycle].pPointMove.trsf),x_tTool,x_mDesc)
          endIf
        break
        case 2
          // Z VALUE
          if pt:tTraj[sTrajCycle].fFrame.trsf!={0,0,0,0,0,0}
            l_pHere=here(x_tTool,pt:tTraj[sTrajCycle].fFrame)
            l_pHere.trsf.z=pt:tTraj[sTrajCycle].pPointMove.trsf.z
            if x_nMoveType==0
              x_nMoveId=movej(l_pHere,x_tTool,x_mDesc)
            elseIf x_nMoveType==1
              x_nMoveId=movel(l_pHere,x_tTool,x_mDesc)
            endIf
          endIf
        break
        case 3,4
          // @POINT @JPOINT
          call getJointData(l_jMove,l_tTool,x_bCycle,x_nIndex)
          // MOVE
          if x_nMoveType==0
            x_nMoveId=movej(l_jMove,x_tTool,x_mDesc)
          elseIf x_nMoveType==1
            l_pPoint=jointToPoint(x_tTool,world,l_jMove)
            l_pPoint.config={ssame,esame,wsame}
            x_nMoveId=movel(l_pPoint,x_tTool,x_mDesc)
          endIf
        break
      endSwitch
    else
      // get the JOINT DATA
      call getJointData(l_jMove,l_tTool,x_bCycle,x_nIndex)
      // MOVE
      if x_nMoveType==0
        x_nMoveId=movej(l_jMove,l_tTool,x_mDesc)
      elseIf x_nMoveType==1
        l_pPoint=jointToPoint(l_tTool,world,l_jMove)
        l_pPoint.config={ssame,esame,wsame}
        x_nMoveId=movel(l_pPoint,l_tTool,x_mDesc)
      endIf
    endIf
  else
    //
    // go to the select Joint
    //
    // use the go to the defined type...
    if x_nIndex==0 and jEditPoint.nZoneType!=0
      switch jEditPoint.nZoneMove
        // POINT TO
        case 0
          if x_nMoveType==0
            x_nMoveId=movej(jEditPoint.pPointMove,x_tTool,x_mDesc)
          elseIf x_nMoveType==1
            x_nMoveId=movel(jEditPoint.pPointMove,x_tTool,x_mDesc)
          endIf
        break
        case 1
          // APPRO gat the tool taught
          call tcp:getTool(l_tTool,jEditPoint.nIndexTool)
          if x_nMoveType==0
            x_nMoveId=movej(appro(here(l_tTool,world),jEditPoint.pPointMove.trsf),x_tTool,x_mDesc)
          elseIf x_nMoveType==1
            x_nMoveId=movel(appro(here(l_tTool,world),jEditPoint.pPointMove.trsf),x_tTool,x_mDesc)
          endIf
        break
        case 2
          // Z VALUE
          if jEditPoint.fFrame.trsf!={0,0,0,0,0,0}
            l_pHere=here(x_tTool,jEditPoint.fFrame)
            l_pHere.trsf.z=jEditPoint.pPointMove.trsf.z
            if x_nMoveType==0
              x_nMoveId=movej(l_pHere,x_tTool,x_mDesc)
            elseIf x_nMoveType==1
              x_nMoveId=movel(l_pHere,x_tTool,x_mDesc)
            endIf
          endIf
        break
        case 3,4
          // get the JOINT DATA
          call getJointData(l_jMove,l_tTool,x_bCycle,x_nIndex)
          // MOVE
          if x_nMoveType==0
            x_nMoveId=movej(l_jMove,x_tTool,x_mDesc)
          elseIf x_nMoveType==1
            l_pPoint=jointToPoint(x_tTool,world,l_jMove)
            l_pPoint.config={ssame,esame,wsame}
            x_nMoveId=movel(l_pPoint,x_tTool,x_mDesc)
          endIf
        break
      endSwitch
    else
      // get the JOINT DATA
      call getJointData(l_jMove,l_tTool,x_bCycle,x_nIndex)
      // MOVE
      if x_nMoveType==0
        x_nMoveId=movej(l_jMove,l_tTool,x_mDesc)
      elseIf x_nMoveType==1
        l_pPoint=jointToPoint(l_tTool,world,l_jMove)
        l_pPoint.config={ssame,esame,wsame}
        x_nMoveId=movel(l_pPoint,l_tTool,x_mDesc)
      endIf
    endIf
  endIf
end

--- new.pgx ---
public program new(string x_sName, num& x_nResult[])
  local string l_sPrefix
  local num l_nResult
begin
  // new one
  if insert(pt:tTraj[x_sName])
    call pt:link_it(x_sName)
    pt:tTraj[x_sName].nIndexTool=saveData:nIndexTool
    x_nResult=0
    // set it
    bToSave=true
  else
    x_nResult=-1
  endIf
end

--- onEdit.pgx ---
public program onEdit(string& x_sItem[])
  local string l_sPath
  local string l_sName
  local num l_nResult
begin
  // DEFINE YOUR ITEM
  call getTrajType(saveData:sTrajTypeUsing)
  // load the trajectory
  call load(x_sItem,l_nResult)
  if size(x_sItem)>1
    // give back the path
    l_sPath="Disk://trajectory/page_viewTraj"
    x_sItem[1]=x_sItem
    x_sItem=l_sPath
    // init
    tAppro={0,0,0,0,0,0}
    tPointTo={0,0,0,0,0,0}
    nZeta=0
  endIf
end

--- onEditItem.pgx ---
public program onEditItem(string& x_sEvent[], num x_nIndex, num x_nIndexItem)
  local joint l_jJoint
  local num i
  local string l_sMessage
  local string l_sEmpty
  local string l_sItem5[5]
  local num l_nMin
  local num l_nMax
  local num l_nValue
  local trsf l_tNull
  local tool l_tTool
  local point l_pPoint
  local num l_nSize
  local num l_nKey
  local num l_nIndex
  local string l_sEvent
  local string l_sItem[4]
begin
  // edit the custom element that was add in the list
  l_jJoint=jEditPoint.tData[x_nIndexItem].jJoint
  call use:findPos(x_sEvent,">",i)
  i=i+1
  // clean the line
  call use:listcursor(use:nView,false)
  l_sEmpty=""
  if x_nIndexItem>0 or (jEditPoint.nZoneType[x_nIndexItem]==0)
    if find(jEditPoint.tData[x_nIndexItem].tSuper.comment,"@")==-1 and (jEditPoint.nZoneType==0 or x_nIndexItem>0)
      switch x_nIndex
        case 0
          //  j1-value
          if cycleStatus:bCycle
            // set a limit +- 5
            call use:changeValue(l_jJoint.j1,l_jJoint.j1-5,l_jJoint.j1+5,i+40-use:nBottomX,use:nView+1,l_sEmpty)
          else
            call use:changeValue(l_jJoint.j1,0,0,i+40-use:nBottomX,use:nView+1,l_sEmpty)
          endIf
        break
        case 1
          //  j2-value
          if cycleStatus:bCycle
            // set a limit +- 5
            call use:changeValue(l_jJoint.j2,l_jJoint.j2-5,l_jJoint.j2+5,i+40-use:nBottomX,use:nView+1,l_sEmpty)
          else
            call use:changeValue(l_jJoint.j2,0,0,i+40-use:nBottomX,use:nView+1,l_sEmpty)
          endIf
        break
        case 2
          //  j3-value
          if cycleStatus:bCycle
            // set a limit +- 5
            call use:changeValue(l_jJoint.j3,l_jJoint.j3-5,l_jJoint.j3+5,i+40-use:nBottomX,use:nView+1,l_sEmpty)
          else
            call use:changeValue(l_jJoint.j3,0,0,i+40-use:nBottomX,use:nView+1,l_sEmpty)
          endIf
        break
        case 3
          //  j4-value
          if cycleStatus:bCycle
            // set a limit +- 5
            call use:changeValue(l_jJoint.j4,l_jJoint.j4-5,l_jJoint.j4+5,i+40-use:nBottomX,use:nView+1,l_sEmpty)
          else
            call use:changeValue(l_jJoint.j4,0,0,i+40-use:nBottomX,use:nView+1,l_sEmpty)
          endIf
        break
        case 4
          //  j5-value
          if cycleStatus:bCycle
            // set a limit +- 5
            call use:changeValue(l_jJoint.j5,l_jJoint.j5-5,l_jJoint.j5+5,i+40-use:nBottomX,use:nView+1,l_sEmpty)
          else
            call use:changeValue(l_jJoint.j5,0,0,i+40-use:nBottomX,use:nView+1,l_sEmpty)
          endIf
        break
        case 5
          //  j6-value
          if cycleStatus:bCycle
            // set a limit +- 5
            call use:changeValue(l_jJoint.j6,l_jJoint.j6-5,l_jJoint.j6+5,i+40-use:nBottomX,use:nView+1,l_sEmpty)
          else
            call use:changeValue(l_jJoint.j6,0,0,i+40-use:nBottomX,use:nView+1,l_sEmpty)
          endIf
        break
      endSwitch
    endIf
    switch x_nIndex
      case 6
        // change the move type
        l_sItem="---"
        l_sItem[1]="Box"
        l_sItem[2]="Sphere"
        l_sItem[3]="Plane"
        call use:clear(0,13)
        call use:changeValue(jEditPoint.nZoneType[x_nIndexItem],0,0,i+40-use:nBottomX,use:nView+1,l_sItem)
      break
    endSwitch
  elseIf x_nIndexItem==0
    switch x_nIndex
      // change the MOVE-TYPE
      case 0
        l_sItem[0]=" - - - "
        l_sItem[1]="Box"
        l_sItem[2]="Sphere"
        l_sItem[3]="Plane"
        call use:clear(0,13)
        call use:changeValue(jEditPoint.nZoneType,0,0,i+40-use:nBottomX,use:nView+1,l_sItem)
      break
      // edit the MOVE-TYPE
      case 1
        switch jEditPoint.nZoneType
          case 1
            // BOX
            call setPointFrame(jEditPoint.fFrame.trsf,jEditPoint.pO,jEditPoint.pX,jEditPoint.pY,jEditPoint.nDimension,1)
            if jEditPoint.fFrame.trsf=={0,0,0,0,0,0}
              call use:timerDialog("the frame has NOT been teached",2)
            endIf
          break
          case 2
            // sphere
            call page_changeTrsf(jEditPoint.pO.trsf,"Sphere"," teach the origin...",true,jEditPoint.nDimension,"radius",world)
            jEditPoint.pX=compose(jEditPoint.pO,world,{100,0,0,0,0,0})
            jEditPoint.pY=compose(jEditPoint.pO,world,{0,100,0,0,0,0})
            setFrame(jEditPoint.pO,jEditPoint.pX,jEditPoint.pY,jEditPoint.fFrame)
          break
          case 3
            //plane
            call setPointFrame(jEditPoint.fFrame.trsf,jEditPoint.pO,jEditPoint.pX,jEditPoint.pY,jEditPoint.nDimension,3)
            if jEditPoint.fFrame.trsf=={0,0,0,0,0,0}
              call use:timerDialog("the frame has NOT been teached",2)
            endIf
          break
        endSwitch
      break
      // CHANGE THE MOVE-TO
      case 2
        // change the move to
        l_sItem5[0]="Point"
        l_sItem5[1]="Appro"
        l_sItem5[2]="Z value"
        //l_sItem5[3]="@JPoint"
        //l_sItem5[4]="@Point"
        call use:clear(0,13)
        // change it
        l_nValue=jEditPoint.nZoneMove
        // sphere has not coord Z movement
        if jEditPoint.nZoneMove==2
          l_sItem5[2]=""
        endIf
        call use:changeValue(jEditPoint.nZoneMove,0,0,i+40-use:nBottomX,use:nView+1,l_sItem5)
        // patch for the sphere
        if jEditPoint.nZoneMove==2 and l_nValue>=2
          l_nValue=l_nValue+1
        endIf
        if l_nValue!=jEditPoint.nZoneMove
          switch jEditPoint.nZoneMove
            case 0
              // reset ?
              if tPointTo=={0,0,0,0,0,0}
                jEditPoint.pPointMove.trsf=tPointTo
              endIf
            break
            case 1
              // reset ?
              if tAppro=={0,0,0,0,0,0}
                jEditPoint.pPointMove.trsf=tAppro
              endIf
            break
            case 2
              // reset ?
              if nZeta==0
                jEditPoint.pPointMove.trsf={0,0,-nZeta,0,0,0}
              endIf
            break
            case 3
              // @Point
              jEditPoint.tData.tSuper.comment=""
            break
            case 4
              // @JPoint
              jEditPoint.tData.tSuper.comment=""
            break
          endSwitch
        endIf
      break
      // EDIT THE MOVE-TO
      case 3
        switch jEditPoint.nZoneMove
          case 0
            // Point
            if tPointTo=={0,0,0,0,0,0}
              tPointTo=jEditPoint.pPointMove.trsf
            endIf
            if (jEditPoint.nZoneType==2 or setFrame(jEditPoint.pO,jEditPoint.pX,jEditPoint.pY,jEditPoint.fFrame)==0)
              call page_changeTrsf(tPointTo,"Point TO"," ",true,jEditPoint.nDimension,"",jEditPoint.fFrame)
              // validate
              if tPointTo!=jEditPoint.pPointMove.trsf
                jEditPoint.pPointMove.trsf=tPointTo
              endIf
            else
              call use:timerDialog("Frame is not Defined ! ",2)
            endIf
          break
          case 1
            // Appro
            if tAppro=={0,0,0,0,0,0}
              tAppro=jEditPoint.pPointMove.trsf
            endIf
            call page_changeTrsf(tAppro,"Appro"," ",false,jEditPoint.nDimension,"",jEditPoint.fFrame)
            // validate
            if tAppro!=jEditPoint.pPointMove.trsf
              jEditPoint.pPointMove.trsf=tAppro
            endIf
          break
          case 2
            // Z Value
            l_nMin=-500
            l_nMax=500
            l_sMessage="coord. Z "
            if nZeta==0
              nZeta=jEditPoint.pPointMove.trsf.z
            endIf
            // edit
            l_nValue=nZeta
            call use:editNumField("Move to a fix Z value",l_sMessage,l_nValue,l_nMin,l_nMax)
            // validate
            if nZeta!=l_nValue
              nZeta=l_nValue
              jEditPoint.pPointMove.trsf.z=l_nValue
            endIf
          break
          //          case 3,4
          //            // select the @Point - @jPoint
          //            // build the list
          //            call use:setSizeList(0,0,16,12)
          //            if jEditPoint.nZoneMove==4
          //              // POINT
          //              call use:listcreate("@Point")
          //              // insert all the item
          //              l_sItem=first(pPoint:pCollection)
          //              call use:listadd(l_sItem)
          //              // search it
          //              while l_sItem!=""
          //                l_sItem=next(pPoint:pCollection[l_sItem])
          //                call use:listadd(l_sItem)
          //                delay(0)
          //              endWhile
          //              l_sItem="@POINT "
          //            elseIf jEditPoint.nZoneMove==3
          //              // JPOINT
          //              call use:listcreate("@JPoint")
          //              // insert all the item
          //              l_sItem=first(jPoint:tTraj)
          //              call use:listadd(l_sItem)
          //              // search it
          //              while l_sItem!=""
          //                l_sItem=next(jPoint:tTraj[l_sItem])
          //                call use:listadd(l_sItem)
          //              endWhile
          //              l_sItem="@JPOINT "
          //            endIf
          //            // refresh it
          //            call use:listupdate(0)
          //            // get the item
          //            do
          //              l_nKey=get()
          //              call use:listevent(l_nKey,l_nIndex,l_sEvent)
          //            until l_nKey==270 or l_nKey==255
          //            // give back
          //            if l_nKey==270
          //              jEditPoint.tData.tSuper.comment=l_sItem+l_sEvent
          //            endIf
          //          break
        endSwitch
      break
    endSwitch
  endIf
  //
  if isInRange(l_jJoint)
    jEditPoint.tData[x_nIndexItem].jJoint=l_jJoint
  else
    // error using the trsf
    call language:message(l_sMessage,-5)
    popUpMsg(l_sMessage)
  endIf
  // wait no key
  call use:nullKey(nKey)
end

--- onFunctionEdit.pgx ---
public program onFunctionEdit(num x_nIndex, string x_sEvent, num x_nFunctionKey)
  local string l_sMessage
  local bool l_bYes
  local string l_sButton[2]
  local string l_sItem
  local tool l_tTool
  local point l_pAlign
  local string l_sMessage2
  local string l_sPage
begin
  //
  // do on Key action
  //
  // x_nIndex = actual index item
  // x_sEvent = actual event item
  //
  switch x_nFunctionKey
    // F1 button
    case 271
      // HERE JOINT
      if !cycleStatus:bCycle and find(jEditPoint.tData[x_nIndex].tSuper.comment,"@")==-1
        call language:message(l_sMessage,160)
        call language:getYesNo(l_sButton)
        // ask the yes_no question
        call use:yes_no(l_sMessage,l_sButton,l_bYes)
        if l_bYes
          call HerePoint(x_nIndex)
        endIf
      endIf
    break
    // F2 button
    case 272
      // ALIGN
      if !cycleStatus:bCycle
        resetMotion()
        // tool
        call tcp:getTool(l_tTool,jEditPoint.nIndexTool)
        l_pAlign=here(l_tTool,world)
        l_pAlign.trsf=align(l_pAlign.trsf,saveData:fFrameItem[saveData:nFrameActive].fFrame.trsf)
        call language:message(l_sMessage,203)
        call language:message(l_sMessage2,134)
        l_sMessage=l_sMessage+" "+l_sMessage2+"..."
        call use:timerDialog(l_sMessage,0)
        movej(l_pAlign,l_tTool,mMdesc)
        watch(isEmpty() or isKeyPressed(255),3)
        if !isEmpty()
          resetMotion()
        endIf
        delay(2)
      endIf
    break
    // F3 button
    case 273
      // Select the gun
      l_sPage="Disk://kernel/page/tool"
      call loadPage(l_sPage,l_sItem)
      // set the tool
      jEditPoint.nIndexTool=saveData:nIndexTool
    break
    // F4 button
    case 274
    break
    // F5 button
    case 275
    break
    // F6 button
    case 276
    break
    // F7 button
    case 277
    break
    // F8 button
    case 278
    break
  endSwitch
end

--- onFunctionSel.pgx ---
public program onFunctionSel(num x_nIndex, string x_sEvent, num x_nFunctionKey)
  local string l_sMessage
  local string l_sMessage2
  local string l_sSwap
  local num l_nResult
  local bool l_bYes
  local string l_sPath
  local string l_sButton[2]
  local string l_sItem
  local num l_nX
  local num l_nY
  local string l_sString
  local string l_sName
begin
  //
  // do on Key action
  //
  // x_nIndex = actual index item
  // x_sEvent = actual event item
  //
  l_nX=40-use:nBottomX-1
  l_nY=use:nBottomY+1
  switch x_nFunctionKey
    // F1 button
    case 271
    break
    // F2 button
    case 272
    break
    // F3 button
    case 273
      //
      // go to the edit program
      //
      l_sPath=prog:libPath()+"/page_instr"
      l_sItem="HOME1"
      call loadPage(l_sPath,l_sItem)
    break
    // F4 button
    case 274
      //
      // go to the edit program
      //
      l_sPath=prog:libPath()+"/page_instr"
      l_sItem="HOME2"
      call loadPage(l_sPath,l_sItem)
    break
    // F5 button
    case 275
    break
    // F6 button
    case 276
    break
    // F7 button
    case 277
      //
      //
      //
    break
    // F8 button
    case 278
    break
  endSwitch
end

--- onFunctionView.pgx ---
public program onFunctionView(num x_nIndex, string x_sEvent, num x_nFunctionKey)
  local string l_sMessage
  local string l_sButton[2]
  local bool l_bYes
  local string l_sItem
  local point l_pAlign
  local tool l_tTool
  local joint l_jJoint
  local string l_sMessage2
  local num l_nIndexFrame
  local frame l_fFrame
begin
  //
  // do on Key action
  //
  // x_nIndex = actual index item
  // x_sEvent = actual event item
  //
  switch x_nFunctionKey
    // F1 button
    case 271
      // HERE JOINT
      if !cycleStatus:bCycle and find(jEditPoint.tData[x_nIndex].tSuper.comment,"@")==-1
        call language:message(l_sMessage,160)
        call language:getYesNo(l_sButton)
        // ask the yes_no question
        call use:yes_no(l_sMessage,l_sButton,l_bYes)
        if l_bYes
          call HerePoint(x_nIndex)
        endIf
      endIf
    break
    // F2 button
    case 272
      // @POINT -> use depart
      // @JOINT -> use the first JOINT
      //call link_me(x_nIndex)
       // ALIGN
      if !cycleStatus:bCycle and !cycleStatus:bSimulation
        resetMotion()
        call getFrameId(l_nIndexFrame)
        l_fFrame=saveData:fFrameItem[l_nIndexFrame].fFrame
        // tool
        call tcp:getTool(l_tTool,jEditPoint.nIndexTool)
        l_pAlign=here(l_tTool,l_fFrame)
        l_pAlign.trsf=align(l_pAlign.trsf,l_fFrame.trsf)
        // check the align
        if pointToJoint(l_tTool,herej(),l_pAlign,l_jJoint)
          call language:message(l_sMessage,203)
          call language:message(l_sMessage2,134)
          l_sMessage=l_sMessage+" "+l_sMessage2+"..."
          call use:timerDialog(l_sMessage,0)
          movej(l_pAlign,l_tTool,mMdesc)
          watch(isEmpty() or isKeyPressed(255),3)
          if !isEmpty()
            resetMotion()
          endIf
          delay(2)
        endIf
      endIf
    break
    // F3 button
    case 273
    break
    // F4 button
    case 274
    break
    // F5 button
    case 275
    break
    // F6 button
    case 276
    break
    // F7 button
    case 277
    break
    // F8 button
    case 278
    break
  endSwitch
  // save the actual index
  nIndex=x_nIndex
end

--- onInsert.pgx ---
public program onInsert(string& x_sItem[])
  local string l_sEvent
  local num l_nKey
  local num l_nIndex
  local num l_nSize
  local num i
begin
  // get the traj type
  x_sItem="home"
end

--- onRun.pgx ---
public program onRun(string& x_sItem[])
  local num l_nSize
  local num l_nResult
  local num i
  local point l_pHere
  local string l_sHome
  local num l_nBest[3]
  local num j
  local string l_sMessage
  local tool l_tTool
  local num l_nJoint
  local joint l_jHere
  local num l_nDistance
  local bool l_bFoundHome
  local string l_sPath
  local num l_nItem
  local bool l_bZoneFound
  local bool l_bInside
  local num l_nJoint4
  local num l_nJoint5
  local num l_nJoint6
  local joint l_jJoint
  local point l_pConfig
  local point l_pCheck
  local joint l_jCheck
begin
  // verify that exist a valid HOME:home
  // do the last home strategy
  call loadCycle("home",l_nResult)
  if pt:tTraj[sTrajCycle].tData[0].jJoint!={0,0,0,0,0,0}
    //
    // inizialize the system
    //
    // reset Distance index home
    l_nItem=-1
    call use:numCopy(l_nItem,nDistance)
    l_nItem=0
    call use:numCopy(l_nItem,nCoeff)
    call use:numCopy(l_nItem,nJoint)
    call use:numCopy(l_nItem,nHome)
    // refresh it
    use:bUseRefresh=true
    // set the start of HOMING
    cycleStatus:bHoming=true
    cycleStatus:bTraj=true
    //
    logMsg("HOMING STRATEGY> RUN ")
    // take the TOOL use flange as template
    l_tTool=flange
    l_pHere=here(flange,world)
    l_jHere=herej()
    // take the size
    call getSize(l_nSize)
    // check for the ZONE
    for i=0 to l_nSize-1
      call get(l_sHome,i)
      if l_sHome!=""
        call loadCycle(l_sHome,l_nResult)
        if l_nResult==0
          pPoints[0]=pt:tTraj[sTrajCycle].pO
          pPoints[1]=pt:tTraj[sTrajCycle].pX
          pPoints[2]=pt:tTraj[sTrajCycle].pY
          // HOME STRATEGY FOR THE ZONE
          call checkZone(pPoints,l_tTool,pt:tTraj[sTrajCycle].nDimension,pt:tTraj[sTrajCycle].nZoneType,l_bInside)
          // check the zone
          if l_bInside
            l_nDistance=distance(pPoints[0],here(l_tTool,world))
            // check if it is the best
            call orderZone(l_nDistance,pt:tTraj[sTrajCycle].nZoneType,i,l_nBest)
            l_bZoneFound=true
          endIf
        endIf
      endIf
    endFor
    if l_bZoneFound
      // save the value to l_nBest
      call selectZone(l_nBest)
      // get the home trajectory
      call get(l_sHome,l_nBest)
      if l_sHome!=""
        // execute the zone strategy
        call loadCycle(l_sHome,l_nResult)
        // execute the trajectory
        if l_nResult==0
          call makeTraj(0,l_sHome)
        else
          call language:message(l_sMessage,-7)
          popUpMsg(l_sMessage+l_sHome+" ; "+toString("",l_nResult))
          logMsg("error on loading "+l_sHome+" ; "+toString("",l_nResult))
        endIf
      endIf
    else
      l_nBest=l_nBest[1]=l_nBest[2]=0
      // find the best point to proced
      for i=0 to l_nSize-1
        // all the traj
        call get(l_sHome,i)
        if l_sHome!=""
          call loadCycle(l_sHome,l_nResult)
          if l_nResult==0
            // HOME STRATEGY FOR THE POINT....
            l_bFoundHome=true
            //
            // STEP 1
            //
            // look for all the joint the best suitable
            for j=0 to size(pt:tTraj[sTrajCycle].tData)-1
              if pt:tTraj[sTrajCycle].nZoneType==0 or j>0
                // check for the best distance
                call getJointData(l_jJoint,l_tTool,true,j)
                // check for the config if not put a big DISTANCE -> 100000
                l_pConfig=jointToPoint(flange,world,l_jJoint)
                if l_pHere.config!=l_pConfig.config and saveData:bUseHomeConfig
                  logMsg("joint: "+toString("",j)+"of the HOME "+l_sHome+" different config ")
                  l_nDistance=100000
                else
                  call scan_bestFit(flange,j,l_pCheck)
                  if !pointToJoint(flange,l_jJoint,l_pCheck,l_jCheck)
                    l_jCheck=l_jJoint
                  endIf
                  l_nDistance=distance(l_pCheck,l_pHere)
                  l_nJoint4=(l_jHere.j4-l_jJoint.j4)*(l_jHere.j4-l_jJoint.j4)
                  l_nJoint5=(l_jHere.j5-l_jJoint.j5)*(l_jHere.j5-l_jJoint.j5)
                  l_nJoint6=(l_jHere.j6-l_jJoint.j6)*(l_jHere.j6-l_jJoint.j6)
                  l_nJoint=sqrt(l_nJoint4+l_nJoint5+l_nJoint6)
                endIf
                l_nBest[2]=l_nDistance
                l_nBest[1]=j
                l_nBest[0]=i
                call orderDistance(l_nBest,l_nJoint)
              endIf
            endFor
          endIf
        endIf
        if l_nResult>0
          logMsg("HOME on RUN> error on loading "+l_sHome+" : "+toString("",l_nResult))
          return
        endIf
      endFor
      // the point has been found
      if l_bFoundHome
        // find the best point
        call select(l_nBest)
        //
        // best Joint Home Trajectory-> l_nBest[0]
        // best Joint Home index     -> l_nBest[1]
        //
        call get(l_sHome,l_nBest[0])
        call loadCycle(l_sHome,l_nResult)
        // execute the trajectory
        if l_nResult==0
          call makeTraj(l_nBest[1],l_sHome)
        else
          call language:message(l_sMessage,-7)
          popUpMsg(l_sMessage+l_sHome+" ; "+toString("",l_nResult))
          logMsg("error on loading "+l_sHome+" ; "+toString("",l_nResult))
        endIf
      endIf
    endIf
    // execute the last HOME trajectory
    if l_sHome!="home"
      // do the last home strategy
      call loadCycle("home",l_nResult)
      // execute the trajectory
      if l_nResult==0 and pt:tTraj[sTrajCycle].tData.jJoint!={0,0,0,0,0,0}
        waitEndMove()
        call makeTraj(0,"home")
        //
      endIf
    endIf
    waitEndMove()
  else
    call language:message(l_sMessage,169)
    popUpMsg(l_sMessage+" HOME JOINT 0,0,0,0,0,0 ")
  endIf
end

--- onSave.pgx ---
public program onSave(string& x_sItem[])
  local num i
  local num l_nSize
  local TrajectoryItem l_tTraj
begin
  //if bToSave
  // update
  if isDefined(pt:tTraj[jEditPoint.sID])
    pt:tTraj[jEditPoint.sID]=jEditPoint
    call pt:link_it(jEditPoint.sID)
    if jEditPoint.sID=="home"
      cycleStatus:bHomeLoaded=false
    endIf
  endIf
  // saveIt
  pt:libSave()
  bToSave=false
  // endIf
end

--- onStart.pgx ---
public program onStart(string& x_sItem[])
  local num i
  local string l_sType
begin
// on START
end

--- onStop.pgx ---
public program onStop(string& x_sItem[])
begin
  if x_sItem=="kill"
    // empty the ram
    pt:libLoad("Disk://kernel/template/session/saveTraj/HOME")
  endIf
end

--- orderDistance.pgx ---
program orderDistance(num& x_nValue[] (dimensions=1), num x_nCoeff (dimensions=1))
  local num l_nValue[4]
  local num i
begin
  //
  // x_nValue[0]= home index
  // x_nValue[1]= joint index
  // x_nValue[2]= nDistance
  // x_nCoeff = coefficent using J4 J5 J6
  //
  // INIT
  //
  // copy
  l_nValue=x_nValue
  l_nValue[1]=x_nValue[1]
  l_nValue[2]=x_nValue[2]
  l_nValue[3]=x_nCoeff
  //
  if nDistance==-1
    nDistance=x_nValue[2]
    nJoint=x_nValue[1]
    nHome=x_nValue
    nCoeff=x_nCoeff
  else
    // MAKE THE  LIST
    for i=0 to size(nDistance)-1
      // a minimum find
      if x_nValue[2]<nDistance[i]
        call insertValue(l_nValue,i)
        return
      else
        // not found put at the end
        if i==size(nDistance)-1
          call insertValue(l_nValue,i+1)
          return
        endIf
      endIf
    endFor
  endIf
end

--- orderZone.pgx ---
program orderZone(num x_nDistance (dimensions=1), num x_nType (dimensions=1), num x_nTrajectory (dimensions=1), num& x_nBest[] (dimensions=1))
  local num l_nValue[4]
  local num i
  local bool l_bFound
begin
  //
  // check if the new HOME trajectory is better then the last one...
  //
  // MOVETYPE PRIORITY
  //
  // BOX -> SPHERE -> PLANE
  //
  // SAME MOVETYPE
  //
  // check the distance from the plane or the center of the sphere
  //
  // x_nTrajectory= home index
  // 0= joint index
  // x_nDistance= nDistance
  // type CUBE-SPHERE-PLANE= nCoeff
  //
  // copy all the value
  l_nValue=x_nTrajectory
  l_nValue[1]=0
  l_nValue[2]=x_nDistance
  l_nValue[3]=x_nType
  // order all
  // MINOR
  if x_nType<nCoeff
    // insert into
    call insertValue(l_nValue,0)
    // EQUAL order by distance
  elseIf x_nType==nCoeff
    // order by distance
    for i=0 to size(nCoeff)-1
      if x_nDistance<=nDistance[i] or i==size(nCoeff)-1
        // insert
        call insertValue(l_nValue,i)
        // exit
        i=size(nCoeff)-1
      endIf
    endFor
    // MAJOR
  elseIf x_nType>nCoeff
    // order by type
    for i=0 to size(nCoeff)-1
      if nCoeff[i]==x_nType
        // found it
        l_bFound=true
        if x_nDistance<=nDistance[i] or i==size(nCoeff)-1
          // insert
          call insertValue(l_nValue,i+1)
          // exit
          i=size(nCoeff)-1
        endIf
        // not the same but the prevoius one was ok
      elseIf l_bFound
        // insert one before
        call insertValue(l_nValue,i)
        // exit
        i=size(nCoeff)-1
        // found in the last item
      elseIf x_nDistance<=nDistance[i] or (i==size(nCoeff)-1)
        if nDistance[0]==-1
          // first item
          call insertValue(l_nValue,i)
        else
          // insert
          call insertValue(l_nValue,i+1)
        endIf
        // exit
        i=size(nCoeff)-1
      endIf
    endFor
  endIf
end

--- page_changeTrsf.pgx ---
public program page_changeTrsf(trsf& x_tTrsf[], string x_sTitle, string x_sComment, bool x_bHere, num& x_nAddon, string x_sAddon, frame x_fFrame)
  local string l_sEvent
  local num l_nIndex
  local num l_nView
  local bool l_bRefresh
  local string l_sMessage
  local trsf l_tTrsf
  local string l_sItem
  local string l_sEmpty
  local point l_pPoint
  local tool l_tTool
  local num l_nAddon
  local num l_nDistanceX
  local num l_nDistanceY
  local bool l_bCheck
  local joint l_jPoint
begin
  logMsg("[KERNEL] INTERFACE:PAGE changeTrsf "+x_sTitle)
  // INIT all
  //call tcp:getTool(l_tTool,jEditPoint.nIndexTool)
  // use the flange
  l_tTool=flange
  l_bRefresh=false
  l_nIndex=0
  l_nView=0
  call use:setSizeList(19,0,19,8)
  call use:setView(false)
  l_tTrsf=x_tTrsf
  //release the button
  call use:nullKey(nKey)
  if !cycleStatus:bCycle and !cycleStatus:bSimulation
    resetMotion()
  endIf
  if x_bHere
    // use the x_fFrame
    l_pPoint=here(l_tTool,x_fFrame)
    l_pPoint.trsf=x_tTrsf
    l_pPoint.config={sfree,efree,wfree}
  endIf
  l_nAddon=x_nAddon
  // set the frame
  do
    cls()
    call use:type(0,12,x_sComment)
    call use:typeMenu(8,"OK")
    if x_bHere
      call language:message(l_sMessage,150)
      call use:typeMenu(1,l_sMessage)
    endIf
    call use:listcreate(x_sTitle)
    l_sItem=("coord  X > "+toString(".2",l_tTrsf.x))
    call use:listadd(l_sItem)
    l_sItem=("coord  Y > "+toString(".2",l_tTrsf.y))
    call use:listadd(l_sItem)
    l_sItem=("coord  Z > "+toString(".2",l_tTrsf.z))
    call use:listadd(l_sItem)
    l_sItem=("coord RX > "+toString(".2",l_tTrsf.rx))
    call use:listadd(l_sItem)
    l_sItem=("coord RY > "+toString(".2",l_tTrsf.ry))
    call use:listadd(l_sItem)
    l_sItem=("coord RZ > "+toString(".2",l_tTrsf.rz))
    call use:listadd(l_sItem)
    // check for the addon for the sphere
    if x_sAddon!=""
      l_sMessage=x_sAddon+"> "+toString("",l_nAddon)
      call use:listadd(l_sMessage)
    endIf
    // show the list
    use:nView=l_nIndex
    call use:listupdate(l_nIndex-l_nView)
    do
      l_nView=use:nView
      nKey=getKey()
      l_pPoint.trsf=l_tTrsf
      if x_bHere and isEmpty() and pointToJoint(l_tTool,herej(),l_pPoint,l_jPoint) and cycleStatus:nWorkingMode==1
        movej(l_pPoint,l_tTool,{25,25,25,9999,9999,off,50,50})
      endIf
      call use:listevent(nKey,l_nIndex,l_sEvent)
      switch nKey
        case 270
          //
          // clean the line
          call use:listcursor(use:nView,false)
          l_sEmpty=""
          switch l_nIndex
            case 0
              //  x-value
              call use:changeValue(l_tTrsf.x,0,0,10+40-use:nBottomX,use:nView+1,l_sEmpty)
            break
            case 1
              //  y-value
              call use:changeValue(l_tTrsf.y,0,0,10+40-use:nBottomX,use:nView+1,l_sEmpty)
            break
            case 2
              //  z-value
              call use:changeValue(l_tTrsf.z,0,0,10+40-use:nBottomX,use:nView+1,l_sEmpty)
            break
            case 3
              //  rx-value
              call use:changeValue(l_tTrsf.rx,0,0,10+40-use:nBottomX,use:nView+1,l_sEmpty)
            break
            case 4
              //  ry-value
              call use:changeValue(l_tTrsf.ry,0,0,10+40-use:nBottomX,use:nView+1,l_sEmpty)
            break
            case 5
              //  rz-value
              call use:changeValue(l_tTrsf.rz,0,0,10+40-use:nBottomX,use:nView+1,l_sEmpty)
            break
            case 6
              // addon
              l_nIndex=find(l_sEvent,">")
              call use:changeValue(l_nAddon,0,0,l_nIndex+1+2+use:nTopX,use:nView+use:nTopY+1,l_sEmpty)
            break
          endSwitch
          l_bRefresh=true
          // clean the movement
          if !cycleStatus:bCycle and !cycleStatus:bSimulation
            resetMotion()
          endIf
        break
        case 278
          // VALIDATE
          x_tTrsf=l_tTrsf
        break
        case 271
          // here
          // use the x_fFrame
          l_pPoint=here(l_tTool,x_fFrame)
          l_pPoint.config={sfree,efree,wfree}
          l_tTrsf=l_pPoint.trsf
          l_bRefresh=true
        break
      endSwitch
      // special ADDON for the sphere
      if x_sAddon!=""
        //  SPHERE
        call checkZone(l_pPoint,l_tTool,l_nAddon,2,l_bCheck)
        // check it
        if l_bCheck
          // inside the zone
          call language:message(l_sMessage,225)
        else
          // outside the zone
          call language:message(l_sMessage,226)
        endIf
        call use:typeLen(1,11,l_sMessage,39)
      endIf
      delay(0)
    until l_bRefresh==true or nKey==255 or nKey==278
    // check the refresh
    l_bRefresh=false
  until nKey==255 or nKey==278
  // check the key
  if nKey==278
    // validate
    x_tTrsf=l_tTrsf
    x_nAddon=l_nAddon
  endIf
  // release the resource
  call use:nullKey(nKey)
  if !cycleStatus:bCycle and !cycleStatus:bSimulation
    resetMotion()
  endIf
end

--- scan_bestFit.pgx ---
program scan_bestFit(tool x_tTool, num x_nIndex, point& x_pBestFit[])
  local num i
  local bool l_bPrevious
  local bool l_bNext
  local point l_pCheck
  local point l_pHere
  local num l_nSize
  local num l_nDistanceNext
  local num l_nDistancePrev
  local num l_nStopPrev
  local num l_nStopNext
  local num i_from
  local num i_to
  local bool l_bOk
  local num l_nMoveType
  local joint l_jResult
  local joint l_jJoint[3]
begin
  // save the point
  // pBestFit [0] -> previous
  // pBestFit [1] -> actual
  // pBestFit [2] -> next
  // scan all
  call getSizeItem(true,l_nSize)
  l_nDistanceNext=10000
  l_nDistancePrev=10000
  call getMoveType(l_nMoveType,x_nIndex,true)
  // search the three point
  if x_nIndex>0
    l_bPrevious=true
    call getJointData(l_jJoint[0],x_tTool,true,x_nIndex-1)
    x_tTool=flange
    pBestFit[0]=jointToPoint(x_tTool,world,l_jJoint[0])
  endIf
  if x_nIndex<l_nSize-1 and l_nSize>1
    l_bNext=true
    call getJointData(l_jJoint[2],x_tTool,true,x_nIndex+1)
    pBestFit[2]=jointToPoint(x_tTool,world,l_jJoint[2])
  endIf
  call getJointData(l_jJoint[1],x_tTool,true,x_nIndex)
  pBestFit[1]=jointToPoint(x_tTool,world,l_jJoint[1])
  // look if the next point if is better
  if l_bNext
    if setFrame(pBestFit[1],pBestFit[2],pNull,fFrame)==0
      pCheck=here(x_tTool,fFrame)
      if pCheck.trsf.x>=0
        // scan it
        l_pCheck=pBestFit[1]
        l_pHere=here(x_tTool,world)
        // check the nearest point
        for i=0 to 0.4 step 0.1
          if l_nMoveType==0
            call interpolateJ(l_jJoint[1],l_jJoint[2],i,l_jResult,l_bOk)
            l_pCheck=jointToPoint(x_tTool,world,l_jResult)
          else
            l_pCheck.trsf=interpolateL(pBestFit[1].trsf,pBestFit[2].trsf,i)
            l_bOk=true
          endIf
          if l_nDistanceNext>=distance(l_pCheck,l_pHere) and l_bOk
            l_nDistanceNext=distance(l_pCheck,l_pHere)
            //save the value
            l_nStopNext=i
          endIf
        endFor
        // closer search
        i_from=(max(l_nStopNext-0.05,0))
        i_to=(min(l_nStopNext+0.05,1))
        for i=i_from to i_to step 0.01
          if l_nMoveType==0
            call interpolateJ(l_jJoint[1],l_jJoint[2],i,l_jResult,l_bOk)
            l_pCheck=jointToPoint(x_tTool,world,l_jResult)
          else
            l_pCheck.trsf=interpolateL(pBestFit[1].trsf,pBestFit[2].trsf,i)
            l_bOk=true
          endIf
          if l_nDistanceNext>=distance(l_pCheck,l_pHere) and l_bOk
            l_nDistanceNext=distance(l_pCheck,l_pHere)
            //save the value
            l_nStopNext=i
          endIf
        endFor
      endIf
    endIf
  endIf
  // look if there is a previous point
  if l_bPrevious
    if setFrame(pBestFit[0],pBestFit[1],pNull,fFrame)==0
      pCheck=here(x_tTool,fFrame)
      // scan it
      if pCheck.trsf.x>=0
        // scan it
        l_pCheck=pBestFit[1]
        l_pHere=here(x_tTool,world)
        // check the nearest point
        for i=0.6 to 1 step 0.1
          if l_nMoveType==0
            call interpolateJ(l_jJoint[0],l_jJoint[1],i,l_jResult,l_bOk)
            l_pCheck=jointToPoint(x_tTool,world,l_jResult)
          else
            l_pCheck.trsf=interpolateL(pBestFit[0].trsf,pBestFit[1].trsf,i)
            l_bOk=true
          endIf
          if l_nDistancePrev>=distance(l_pCheck,l_pHere)
            l_nDistancePrev=distance(l_pCheck,l_pHere)
            //save the value
            l_nStopPrev=i
          endIf
        endFor
        // closer search
        i_from=(max(l_nStopPrev-0.05,0))
        i_to=(min(l_nStopPrev+0.05,1))
        for i=i_from to i_to step 0.01
          if l_nMoveType==0
            call interpolateJ(l_jJoint[0],l_jJoint[1],i,l_jResult,l_bOk)
            l_pCheck=jointToPoint(x_tTool,world,l_jResult)
          else
            l_pCheck.trsf=interpolateL(pBestFit[0].trsf,pBestFit[1].trsf,i)
            l_bOk=true
          endIf
          if l_nDistancePrev>=distance(l_pCheck,l_pHere)
            l_nDistancePrev=distance(l_pCheck,l_pHere)
            //save the value
            l_nStopPrev=i
          endIf
        endFor
      endIf
    endIf
  endIf
  // go to an approach POINT
  if l_nStopNext!=0 or l_nStopPrev!=0
    if l_nDistanceNext<l_nDistancePrev
      if l_nMoveType==0
        call interpolateJ(l_jJoint[1],l_jJoint[2],l_nStopNext,l_jResult,l_bOk)
        l_pCheck=jointToPoint(x_tTool,world,l_jResult)
      else
        l_pCheck.trsf=interpolateL(pBestFit[1].trsf,pBestFit[2].trsf,l_nStopNext)
      endIf
    else
      if l_nMoveType==0
        call interpolateJ(l_jJoint[0],l_jJoint[1],l_nStopPrev,l_jResult,l_bOk)
        l_pCheck=jointToPoint(x_tTool,world,l_jResult)
      else
        ? l_nStopPrev
        l_pCheck.trsf=interpolateL(pBestFit[0].trsf,pBestFit[1].trsf,l_nStopPrev)
      endIf
    endIf
    // save it
    x_pBestFit=l_pCheck
  else
    // return the default
    x_pBestFit=pBestFit[1]
  endIf
end

--- select.pgx ---
program select(num& x_nSelect[])
  local num i
  local num l_nIndex
  local num l_nMin
begin
  //
  // to save:
  // x_nBest [0] -# Traejctory
  // x_nBest [1] -# index
  //
  // STRATEGY look the FIRST VALUE
  if nDistance>saveData:nRadiusHome
    // take the first
    l_nIndex=0
  else
    // look for the point beyond the radius
    l_nMin=100000
    for i=0 to size(nDistance)-1
      if nDistance[i]<saveData:nRadiusHome
        if nCoeff[i]<l_nMin and abs(nCoeff[i]-l_nMin)>30
          l_nMin=nCoeff[i]
          l_nIndex=i
          if saveData:bDebug
            ? "searching inside"
            ? nDistance[i]
            ? nJoint[i]
            ? nHome[i]
          endIf
        endIf
      else
        // exit
        i=size(nDistance)-1
      endIf
    endFor
  endIf
  // save the value
  x_nSelect[0]=nHome[l_nIndex]
  x_nSelect[1]=nJoint[l_nIndex]
end

--- selectProg.pgx ---
program selectProg(string x_sProg)
  local num l_nSize
  local string l_sEvent
  local num i
  local num l_nIndex
  local string l_sProg
  local num l_nKey
  local string l_sEmpty
begin
  // show the proram list
  call use:clear(0,13)
  //
  call use:stringCopy(l_sEmpty,sList)
  nSelected=-1
  //
  // Build the list
  //
  call prog:getSize(l_nSize)
  for i=0 to l_nSize-1
    call prog:get(l_sEvent,i)
    if l_sEvent!=""
      call listAdd(l_sEvent)
      if l_sEvent==x_sProg
        // select the default
        nSelected=i
      endIf
    endIf
  endFor
  //
  // Show the list
  //
  // define your list size for default
  call use:setSizeList(10,0,17,10)
  //
  call use:listcreate("PROG")
  call use:listadd(sList)
  call use:selectNewField(nSelected,0,0)
  //
  call use:type(35,13,"RESET")
  do
    l_nKey=get()
    call use:listevent(l_nKey,l_nIndex,l_sProg)
    if l_nKey==278
      jEditPoint.sProgram=""
      return
    endIf
  until l_nKey==255 or l_nKey==270
  // save the data
  if l_nKey!=255
    jEditPoint.sProgram=l_sProg
  endIf
end

--- selectZone.pgx ---
program selectZone(num& x_nSelect[] (dimensions=1))
  local num i
  local num l_nIndex
  local num l_nMin
begin
  //
  // to save:
  // x_nBest [0] -# Traejctory
  // x_nBest [1] -# index
  // x_nBest [2] -# Type
  //
  // save the value
  //
  // use the first value
  //
  x_nSelect[0]=nHome[0]
  x_nSelect[1]=0
  x_nSelect[2]=nCoeff[0]
end

--- setFrameId.pgx ---
public program setFrameId(num x_nIndex)
begin
  //
  jEditPoint.nIndexFrame=x_nIndex
end

--- setPointFrame.pgx ---
program setPointFrame(trsf& x_trsfFrame[], point& x_pO, point& x_pX, point& x_pY, num& x_nDimension, num x_nType)
  local string l_sMessage[3]
  local num l_nStep
  local string l_sButton[8]
  local num l_nResult
  local tool l_tTool
  local point l_pHere
  local bool l_bUnreachable
  local num l_nDimension
  local string l_sEmpty
  local num l_nDistanceX
  local num l_nDistanceY
  local point l_pPoint
  local num l_nOldLine
  local joint l_jPoint
  local bool l_bCheck
  local string l_sEvent
  local bool l_bGoto
  local trsf l_tNull
begin
  //
  //  Change the Frame associate to the Trajectory
  //
  cls()
  //
  // copy from saveData
  //
  pPoints[0]=x_pO
  pPoints[1]=x_pX
  pPoints[2]=x_pY
  // use the flange
  l_tTool=flange
  //  call tcp:getTool(l_tTool,jEditPoint.nIndexTool)
  l_nDimension=x_nDimension
  //release the button
  call use:nullKey(nKey)
  //
  do
    call language:message(l_sMessage,150)
    // here
    call language:message(l_sMessage[1],167)
    // put the menu
    call use:typeMenu(1,l_sMessage)
    call use:typeMenu(2,l_sMessage[1])
    // validate
    call use:typeMenu(8,"OK")
    // show the here and the edit button
    call use:setSizeList(21,2,17,5)
    // for the title
    switch x_nType
      case 1
        l_sMessage[2]="BOX"
      break
      case 3
        l_sMessage[2]="PLANE"
      break
    endSwitch
    call use:listcreate(l_sMessage[2])
    //origin
    call language:message(l_sMessage,198)
    // pos. X
    call language:message(l_sMessage[1],199)
    l_sMessage[1]=l_sMessage[1]+" X"
    // pos. Y
    call language:message(l_sMessage[2],199)
    l_sMessage[2]=l_sMessage[2]+" Y"
    call use:listadd(l_sMessage)
    if x_nType==1
      // height for the BOX
      call language:message(l_sMessage[2],224)
      l_sMessage[2]=l_sMessage[2]+"> "+toString("",l_nDimension)
      call use:listadd(l_sMessage[2])
    endIf
    call use:listupdate(0)
    // get the key
    nKey=getKey()
    l_sEmpty=""
    call use:listevent(nKey,l_nResult,l_sEvent)
    //
    if l_nResult!=l_nOldLine or nKey==270
      l_bGoto=true
      l_nOldLine=l_nResult
      if !cycleStatus:bCycle and !cycleStatus:bSimulation
        resetMotion()
      endIf
    else
      l_bGoto=false
    endIf
    switch l_nResult
      case 0
        // take the Origin
        if pointToJoint(l_tTool,herej(),pPoints[0],l_jPoint) and cycleStatus:nWorkingMode==1 and l_bGoto
          movej(pPoints[0],l_tTool,{25,25,25,9999,9999,off,50,50})
        endIf
        // the key has been pressed
        if nKey==271
          pPoints[0]=here(l_tTool,world)
          call language:message(l_sMessage,193)
          call use:type(2,3,l_sMessage)
        elseIf nKey==272 or nKey==270
          call language:message(l_sMessage,198)
          call page_changeTrsf(pPoints[0].trsf,l_sMessage,"",false,l_nStep,"",world)
          cls()
        endIf
      break
      case 1
        //take the X Point
        if pointToJoint(l_tTool,herej(),pPoints[1],l_jPoint) and cycleStatus:nWorkingMode==1 and l_bGoto
          movej(pPoints[1],l_tTool,{25,25,25,9999,9999,off,50,50})
        endIf
        // key pressure
        if nKey==271
          pPoints[1]=here(l_tTool,world)
          call language:message(l_sMessage,193)
          call use:type(2,4,l_sMessage)
        elseIf nKey==272 or nKey==270
          call language:message(l_sMessage,199)
          call page_changeTrsf(pPoints[1].trsf,l_sMessage+" X","",false,l_nStep,"",world)
          cls()
        endIf
      break
      case 2
        // take the Y Point
        if pointToJoint(l_tTool,herej(),pPoints[2],l_jPoint) and cycleStatus:nWorkingMode==1 and l_bGoto
          movej(pPoints[2],l_tTool,{25,25,25,9999,9999,off,50,50})
        endIf
        // key pressure
        if nKey==271
          pPoints[2]=here(l_tTool,world)
          call language:message(l_sMessage,193)
          call use:type(2,5,l_sMessage)
        elseIf nKey==272 or nKey==270
          call language:message(l_sMessage,199)
          call page_changeTrsf(pPoints[2].trsf,l_sMessage+" Y","",false,l_nStep,"",world)
          cls()
        endIf
      break
      case 3
        // modify the Height
        if nKey==270
          l_nStep=find(l_sEvent,">")
          // clean the line
          call use:listcursor(use:nView,false)
          call use:changeValue(l_nDimension,0,0,l_nStep+1+2+use:nTopX,use:nView+use:nTopY+1,l_sEmpty)
        endIf
      break
    endSwitch
    use:nView=l_nResult
    // check the zone
    if setFrame(pPoints[0],pPoints[1],pPoints[2],fSetFrame)==0
      call checkZone(pPoints,l_tTool,l_nDimension,x_nType,l_bCheck)
      // show the result
      if l_bCheck
        // inside the zone
        call language:message(l_sMessage,225)
      else
        //outside the zone
        call language:message(l_sMessage,226)
      endIf
      call use:typeLen(1,11,l_sMessage,39)
    else
      // frame not define
      call language:message(l_sMessage,183)
    endIf
  until nKey==278 or nKey==255
  // check the result
  if nKey==278
    // set the frame
    if setFrame(pPoints[0],pPoints[1],pPoints[2],fSetFrame)==0
      x_trsfFrame=fSetFrame.trsf
      // copy back to save DATA
      x_pO=pPoints[0]
      x_pX=pPoints[1]
      x_pY=pPoints[2]
      x_nDimension=l_nDimension
      //
    else
      call language:message(l_sMessage,183)
      popUpMsg(l_sMessage+toString("",setFrame(pPoints[0],pPoints[1],pPoints[2],fSetFrame)))
    endIf
  endIf
  //release the button
  call use:nullKey(nKey)
end

--- setTrajItem.pgx ---
public program setTrajItem(TrajectoryItem& x_tTraj[], num x_nIndex)
begin
  //
  // set all the field
  //
  jEditPoint.tData[x_nIndex].tSuper=x_tTraj
  // active the save data
  bToSave=true
end
